LIN {X 0,Y 525.412,Z 540.645,A -85,B 0,C 180,E1 -4783.365,E2 -4783.365} C_VEL
LIN {X 0,Y 525.537,Z 527.651,A -85,B 0,C 180,E1 -4783.657,E2 -4783.657} C_VEL
LIN {X 0,Y 525.786,Z 431.838,A -85,B 0,C 180,E1 -4784.981,E2 -4784.981} C_VEL
LIN {X 0,Y 524.311,Z 422.453,A -85,B 0,C 180,E1 -4785.165,E2 -4785.165} C_VEL
LIN {X 0,Y 524.738,Z 402.773,A -85,B 0,C 180,E1 -4788.305,E2 -4788.305} C_VEL
LIN {X 0,Y 525.21,Z 383.773,A -85,B 0,C 180,E1 -4791.385,E2 -4791.385} C_VEL
LIN {X 0,Y 525.337,Z 376.275,A -85,B 0,C 180,E1 -4792.618,E2 -4792.618} C_VEL
LIN {X 0,Y 523.946,Z 368.721,A -85,B 0,C 180,E1 -4793.942,E2 -4793.942} C_VEL
LIN {X 0,Y 523.978,Z 368.713,A -85,B 0,C 180,E1 -4796.271,E2 -4796.271} C_VEL
LIN {X 0,Y 523.958,Z 368.72,A -85,B 0,C 180,E1 -4799.324,E2 -4799.324} C_VEL
LIN {X 0,Y 523.943,Z 368.716,A -85,B 0,C 180,E1 -4802.449,E2 -4802.449} C_VEL
LIN {X 0,Y 523.927,Z 368.724,A -85,B 0,C 180,E1 -4805.226,E2 -4805.226} C_VEL
LIN {X 0,Y 523.919,Z 368.718,A -85,B 0,C 180,E1 -4808.102,E2 -4808.102} C_VEL
LIN {X 0,Y 523.961,Z 368.717,A -85,B 0,C 180,E1 -4811.311,E2 -4811.311} C_VEL
LIN {X 0,Y 523.959,Z 368.719,A -85,B 0,C 180,E1 -4814.691,E2 -4814.691} C_VEL
LIN {X 0,Y 523.959,Z 368.713,A -85,B 0,C 180,E1 -4817.882,E2 -4817.882} C_VEL
LIN {X 0,Y 523.923,Z 368.725,A -85,B 0,C 180,E1 -4820.915,E2 -4820.915} C_VEL
LIN {X 0,Y 523.902,Z 368.72,A -85,B 0,C 180,E1 -4823.825,E2 -4823.825} C_VEL
LIN {X 0,Y 523.944,Z 368.723,A -85,B 0,C 180,E1 -4826.636,E2 -4826.636} C_VEL
LIN {X 0,Y 523.958,Z 368.714,A -85,B 0,C 180,E1 -4829.356,E2 -4829.356} C_VEL
LIN {X 0,Y 523.981,Z 368.714,A -85,B 0,C 180,E1 -4832.281,E2 -4832.281} C_VEL
LIN {X 0,Y 523.951,Z 368.723,A -85,B 0,C 180,E1 -4834.581,E2 -4834.581} C_VEL
LIN {X 0,Y 523.922,Z 368.718,A -85,B 0,C 180,E1 -4837.756,E2 -4837.756} C_VEL
LIN {X 0,Y 523.978,Z 368.718,A -85,B 0,C 180,E1 -4840.408,E2 -4840.408} C_VEL
LIN {X 0,Y 523.97,Z 368.716,A -85,B 0,C 180,E1 -4842.837,E2 -4842.837} C_VEL
LIN {X 0,Y 523.98,Z 368.711,A -85,B 0,C 180,E1 -4845.236,E2 -4845.236} C_VEL
LIN {X 0,Y 524.019,Z 368.715,A -85,B 0,C 180,E1 -4848.394,E2 -4848.394} C_VEL
LIN {X 0,Y 523.993,Z 368.709,A -85,B 0,C 180,E1 -4851.516,E2 -4851.516} C_VEL
LIN {X 0,Y 524.048,Z 368.705,A -85,B 0,C 180,E1 -4853.841,E2 -4853.841} C_VEL
LIN {X 0,Y 524.075,Z 368.7,A -85,B 0,C 180,E1 -4856.925,E2 -4856.925} C_VEL
LIN {X 0,Y 524.119,Z 368.699,A -85,B 0,C 180,E1 -4860,E2 -4860} C_VEL
LIN {X 0,Y 524.076,Z 368.699,A -85,B 0,C 180,E1 -4863.075,E2 -4863.075} C_VEL
LIN {X 0,Y 524.05,Z 368.711,A -85,B 0,C 180,E1 -4866.159,E2 -4866.159} C_VEL
LIN {X 0,Y 524.005,Z 368.711,A -85,B 0,C 180,E1 -4868.484,E2 -4868.484} C_VEL
LIN {X 0,Y 524.007,Z 368.712,A -85,B 0,C 180,E1 -4871.74,E2 -4871.74} C_VEL
LIN {X 0,Y 523.997,Z 368.708,A -85,B 0,C 180,E1 -4875.052,E2 -4875.052} C_VEL
LIN {X 0,Y 523.968,Z 368.721,A -85,B 0,C 180,E1 -4877.969,E2 -4877.969} C_VEL
LIN {X 0,Y 523.976,Z 368.713,A -85,B 0,C 180,E1 -4880.41,E2 -4880.41} C_VEL
LIN {X 0,Y 523.921,Z 368.718,A -85,B 0,C 180,E1 -4882.893,E2 -4882.893} C_VEL
LIN {X 0,Y 523.957,Z 368.717,A -85,B 0,C 180,E1 -4885.419,E2 -4885.419} C_VEL
LIN {X 0,Y 523.973,Z 368.717,A -85,B 0,C 180,E1 -4887.999,E2 -4887.999} C_VEL
LIN {X 0,Y 523.948,Z 368.715,A -85,B 0,C 180,E1 -4890.855,E2 -4890.855} C_VEL
LIN {X 0,Y 523.964,Z 368.721,A -85,B 0,C 180,E1 -4893.735,E2 -4893.735} C_VEL
LIN {X 0,Y 523.925,Z 368.718,A -85,B 0,C 180,E1 -4896.404,E2 -4896.404} C_VEL
LIN {X 0,Y 523.923,Z 368.72,A -85,B 0,C 180,E1 -4899.085,E2 -4899.085} C_VEL
LIN {X 0,Y 523.959,Z 368.715,A -85,B 0,C 180,E1 -4902.119,E2 -4902.119} C_VEL
LIN {X 0,Y 523.959,Z 368.719,A -85,B 0,C 180,E1 -4905.309,E2 -4905.309} C_VEL
LIN {X 0,Y 523.922,Z 368.719,A -85,B 0,C 180,E1 -4906.911,E2 -4906.911} C_VEL
LIN {X 0,Y 523.255,Z 368.809,A -85,B 0,C 180,E1 -4907.553,E2 -4907.553} C_VEL
LIN {X 0,Y 520.412,Z 369.16,A -85,B 0,C 180,E1 -4908.594,E2 -4908.594} C_VEL
LIN {X 0,Y 518.007,Z 369.464,A -85,B 0,C 180,E1 -4909.433,E2 -4909.433} C_VEL
LIN {X 0,Y 516.971,Z 369.585,A -85,B 0,C 180,E1 -4910.081,E2 -4910.081} C_VEL
LIN {X 0,Y 516.885,Z 369.595,A -85,B 0,C 180,E1 -4910.3,E2 -4910.3} C_VEL
LIN {X 0,Y 516.888,Z 369.603,A -85,B 0,C 180,E1 -4913.342,E2 -4913.342} C_VEL
LIN {X 0,Y 516.916,Z 369.591,A -85,B 0,C 180,E1 -4916.121,E2 -4916.121} C_VEL
LIN {X 0,Y 516.894,Z 369.597,A -85,B 0,C 180,E1 -4918.936,E2 -4918.936} C_VEL
LIN {X 0,Y 516.922,Z 369.594,A -85,B 0,C 180,E1 -4921.585,E2 -4921.585} C_VEL
LIN {X 0,Y 516.935,Z 369.59,A -85,B 0,C 180,E1 -4924.211,E2 -4924.211} C_VEL
LIN {X 0,Y 516.868,Z 369.603,A -85,B 0,C 180,E1 -4926.776,E2 -4926.776} C_VEL
LIN {X 0,Y 516.944,Z 369.671,A -85,B 0,C 180,E1 -4928.857,E2 -4928.857} C_VEL
LIN {X 0,Y 517.824,Z 376.138,A -85,B 0,C 180,E1 -4930.166,E2 -4930.166} C_VEL
LIN {X 0,Y 517.497,Z 389.927,A -85,B 0,C 180,E1 -4932.82,E2 -4932.82} C_VEL
LIN {X 0,Y 517.281,Z 399.757,A -85,B 0,C 180,E1 -4934.685,E2 -4934.685} C_VEL
LIN {X 0,Y 519.14,Z 410.322,A -85,B 0,C 180,E1 -4934.899,E2 -4934.899} C_VEL
LIN {X 0,Y 518.727,Z 506.835,A -85,B 0,C 180,E1 -4936.26,E2 -4936.26} C_VEL
LIN {X 0,Y 518.465,Z 520.01,A -85,B 0,C 180,E1 -4936.602,E2 -4936.602} C_VEL
LIN {X 0,Y 518.198,Z 532.106,A -85,B 0,C 180,E1 -4937.069,E2 -4937.069} C_VEL
LIN {X 0,Y 517.99,Z 543.446,A -85,B 0,C 180,E1 -4937.658,E2 -4937.658} C_VEL
LIN {X 0,Y 517.648,Z 555.196,A -85,B 0,C 180,E1 -4938.448,E2 -4938.448} C_VEL
LIN {X 0,Y 517.328,Z 565.677,A -85,B 0,C 180,E1 -4939.333,E2 -4939.333} C_VEL
LIN {X 0,Y 517.077,Z 574.24,A -85,B 0,C 180,E1 -4940.218,E2 -4940.218} C_VEL
LIN {X 0,Y 516.854,Z 582.127,A -85,B 0,C 180,E1 -4941.201,E2 -4941.201} C_VEL
LIN {X 0,Y 516.62,Z 589.84,A -85,B 0,C 180,E1 -4942.378,E2 -4942.378} C_VEL
LIN {X 0,Y 516.458,Z 596.913,A -85,B 0,C 180,E1 -4943.75,E2 -4943.75} C_VEL
LIN {X 0,Y 516.314,Z 601.629,A -85,B 0,C 180,E1 -4944.924,E2 -4944.924} C_VEL
LIN {X 0,Y 516.373,Z 605.238,A -85,B 0,C 180,E1 -4946.098,E2 -4946.098} C_VEL
LIN {X 0,Y 516.282,Z 607.106,A -85,B 0,C 180,E1 -4946.879,E2 -4946.879} C_VEL
LIN {X 0,Y 516.261,Z 608.515,A -85,B 0,C 180,E1 -4947.66,E2 -4947.66} C_VEL
LIN {X 0,Y 516.16,Z 610.136,A -85,B 0,C 180,E1 -4949.22,E2 -4949.22} C_VEL
LIN {X 0,Y 516.155,Z 610.373,A -85,B 0,C 180,E1 -4950,E2 -4950} C_VEL
LIN {X 0,Y 516.16,Z 610.19,A -85,B 0,C 180,E1 -4950.78,E2 -4950.78} C_VEL
LIN {X 0,Y 516.262,Z 608.641,A -85,B 0,C 180,E1 -4952.341,E2 -4952.341} C_VEL
LIN {X 0,Y 516.283,Z 607.286,A -85,B 0,C 180,E1 -4953.122,E2 -4953.122} C_VEL
LIN {X 0,Y 516.363,Z 604.421,A -85,B 0,C 180,E1 -4954.293,E2 -4954.293} C_VEL
LIN {X 0,Y 516.404,Z 600.537,A -85,B 0,C 180,E1 -4955.467,E2 -4955.467} C_VEL
LIN {X 0,Y 516.488,Z 594.693,A -85,B 0,C 180,E1 -4956.812,E2 -4956.812} C_VEL
LIN {X 0,Y 516.669,Z 587.996,A -85,B 0,C 180,E1 -4958.015,E2 -4958.015} C_VEL
LIN {X 0,Y 516.863,Z 579.842,A -85,B 0,C 180,E1 -4959.194,E2 -4959.194} C_VEL
LIN {X 0,Y 517.107,Z 571.496,A -85,B 0,C 180,E1 -4960.177,E2 -4960.177} C_VEL
LIN {X 0,Y 517.464,Z 561.192,A -85,B 0,C 180,E1 -4961.16,E2 -4961.16} C_VEL
LIN {X 0,Y 517.783,Z 549.377,A -85,B 0,C 180,E1 -4962.059,E2 -4962.059} C_VEL
LIN {X 0,Y 518.085,Z 538.006,A -85,B 0,C 180,E1 -4962.735,E2 -4962.735} C_VEL
LIN {X 0,Y 518.364,Z 525.984,A -85,B 0,C 180,E1 -4963.276,E2 -4963.276} C_VEL
LIN {X 0,Y 518.577,Z 512.904,A -85,B 0,C 180,E1 -4963.695,E2 -4963.695} C_VEL
LIN {X 0,Y 518.752,Z 500.391,A -85,B 0,C 180,E1 -4963.94,E2 -4963.94} C_VEL
LIN {X 0,Y 519.037,Z 409.84,A -85,B 0,C 180,E1 -4965.201,E2 -4965.201} C_VEL
LIN {X 0,Y 517.246,Z 399.719,A -85,B 0,C 180,E1 -4965.413,E2 -4965.413} C_VEL
LIN {X 0,Y 517.654,Z 384.021,A -85,B 0,C 180,E1 -4968.401,E2 -4968.401} C_VEL
LIN {X 0,Y 517.769,Z 374.986,A -85,B 0,C 180,E1 -4970.152,E2 -4970.152} C_VEL
LIN {X 0,Y 516.939,Z 369.596,A -85,B 0,C 180,E1 -4971.274,E2 -4971.274} C_VEL
LIN {X 0,Y 516.901,Z 369.6,A -85,B 0,C 180,E1 -4974.361,E2 -4974.361} C_VEL
LIN {X 0,Y 516.928,Z 369.597,A -85,B 0,C 180,E1 -4976.658,E2 -4976.658} C_VEL
LIN {X 0,Y 516.915,Z 369.591,A -85,B 0,C 180,E1 -4979.524,E2 -4979.524} C_VEL
LIN {X 0,Y 516.9,Z 369.598,A -85,B 0,C 180,E1 -4982.543,E2 -4982.543} C_VEL
LIN {X 0,Y 516.873,Z 369.597,A -85,B 0,C 180,E1 -4985.33,E2 -4985.33} C_VEL
LIN {X 0,Y 516.885,Z 369.595,A -85,B 0,C 180,E1 -4987.943,E2 -4987.943} C_VEL
LIN {X 0,Y 516.887,Z 369.602,A -85,B 0,C 180,E1 -4990.742,E2 -4990.742} C_VEL
LIN {X 0,Y 516.887,Z 369.6,A -85,B 0,C 180,E1 -4992.832,E2 -4992.832} C_VEL
LIN {X 0,Y 516.928,Z 369.592,A -85,B 0,C 180,E1 -4995.01,E2 -4995.01} C_VEL
LIN {X 0,Y 516.921,Z 369.597,A -85,B 0,C 180,E1 -4998.399,E2 -4998.399} C_VEL
LIN {X 0,Y 516.885,Z 369.595,A -85,B 0,C 180,E1 -5001.284,E2 -5001.284} C_VEL
LIN {X 0,Y 516.876,Z 369.602,A -85,B 0,C 180,E1 -5004.22,E2 -5004.22} C_VEL
LIN {X 0,Y 516.9,Z 369.593,A -85,B 0,C 180,E1 -5007.053,E2 -5007.053} C_VEL
LIN {X 0,Y 516.897,Z 369.595,A -85,B 0,C 180,E1 -5009.796,E2 -5009.796} C_VEL
LIN {X 0,Y 516.934,Z 369.595,A -85,B 0,C 180,E1 -5012.468,E2 -5012.468} C_VEL
LIN {X 0,Y 516.881,Z 369.595,A -85,B 0,C 180,E1 -5015.07,E2 -5015.07} C_VEL
LIN {X 0,Y 516.874,Z 369.597,A -85,B 0,C 180,E1 -5017.622,E2 -5017.622} C_VEL
LIN {X 0,Y 516.938,Z 369.597,A -85,B 0,C 180,E1 -5020.13,E2 -5020.13} C_VEL
LIN {X 0,Y 516.935,Z 369.591,A -85,B 0,C 180,E1 -5022.596,E2 -5022.596} C_VEL
LIN {X 0,Y 516.949,Z 369.586,A -85,B 0,C 180,E1 -5025.03,E2 -5025.03} C_VEL
LIN {X 0,Y 516.972,Z 369.589,A -85,B 0,C 180,E1 -5028.234,E2 -5028.234} C_VEL
LIN {X 0,Y 516.972,Z 369.585,A -85,B 0,C 180,E1 -5031.4,E2 -5031.4} C_VEL
LIN {X 0,Y 517.017,Z 369.584,A -85,B 0,C 180,E1 -5033.757,E2 -5033.757} C_VEL
LIN {X 0,Y 517.089,Z 369.575,A -85,B 0,C 180,E1 -5037.663,E2 -5037.663} C_VEL
LIN {X 0,Y 517.099,Z 369.568,A -85,B 0,C 180,E1 -5040.779,E2 -5040.779} C_VEL
LIN {X 0,Y 517.019,Z 369.579,A -85,B 0,C 180,E1 -5043.117,E2 -5043.117} C_VEL
LIN {X 0,Y 517.016,Z 369.58,A -85,B 0,C 180,E1 -5046.243,E2 -5046.243} C_VEL
LIN {X 0,Y 516.947,Z 369.591,A -85,B 0,C 180,E1 -5049.389,E2 -5049.389} C_VEL
LIN {X 0,Y 516.99,Z 369.588,A -85,B 0,C 180,E1 -5051.824,E2 -5051.824} C_VEL
LIN {X 0,Y 516.95,Z 369.589,A -85,B 0,C 180,E1 -5055.146,E2 -5055.146} C_VEL
LIN {X 0,Y 516.93,Z 369.59,A -85,B 0,C 180,E1 -5058.222,E2 -5058.222} C_VEL
LIN {X 0,Y 516.918,Z 369.591,A -85,B 0,C 180,E1 -5060.701,E2 -5060.701} C_VEL
LIN {X 0,Y 516.896,Z 369.594,A -85,B 0,C 180,E1 -5064.073,E2 -5064.073} C_VEL
LIN {X 0,Y 516.927,Z 369.59,A -85,B 0,C 180,E1 -5066.658,E2 -5066.658} C_VEL
LIN {X 0,Y 516.916,Z 369.597,A -85,B 0,C 180,E1 -5069.524,E2 -5069.524} C_VEL
LIN {X 0,Y 516.899,Z 369.593,A -85,B 0,C 180,E1 -5072.543,E2 -5072.543} C_VEL
LIN {X 0,Y 516.87,Z 369.604,A -85,B 0,C 180,E1 -5075.329,E2 -5075.329} C_VEL
LIN {X 0,Y 516.884,Z 369.595,A -85,B 0,C 180,E1 -5077.943,E2 -5077.943} C_VEL
LIN {X 0,Y 516.887,Z 369.597,A -85,B 0,C 180,E1 -5080.741,E2 -5080.741} C_VEL
LIN {X 0,Y 516.888,Z 369.599,A -85,B 0,C 180,E1 -5082.831,E2 -5082.831} C_VEL
LIN {X 0,Y 516.927,Z 369.597,A -85,B 0,C 180,E1 -5085.01,E2 -5085.01} C_VEL
LIN {X 0,Y 516.917,Z 369.591,A -85,B 0,C 180,E1 -5088.399,E2 -5088.399} C_VEL
LIN {X 0,Y 516.887,Z 369.599,A -85,B 0,C 180,E1 -5091.284,E2 -5091.284} C_VEL
LIN {X 0,Y 516.877,Z 369.596,A -85,B 0,C 180,E1 -5094.22,E2 -5094.22} C_VEL
LIN {X 0,Y 516.899,Z 369.6,A -85,B 0,C 180,E1 -5097.053,E2 -5097.053} C_VEL
LIN {X 0,Y 516.897,Z 369.595,A -85,B 0,C 180,E1 -5099.796,E2 -5099.796} C_VEL
LIN {X 0,Y 516.93,Z 369.595,A -85,B 0,C 180,E1 -5102.467,E2 -5102.467} C_VEL
LIN {X 0,Y 516.915,Z 369.599,A -85,B 0,C 180,E1 -5105.072,E2 -5105.072} C_VEL
LIN {X 0,Y 516.937,Z 369.68,A -85,B 0,C 180,E1 -5105.903,E2 -5105.903} C_VEL
LIN {X 0,Y 518.386,Z 377.827,A -85,B 0,C 180,E1 -5107.347,E2 -5107.347} C_VEL
LIN {X 0,Y 518.003,Z 392.507,A -85,B 0,C 180,E1 -5109.779,E2 -5109.779} C_VEL
LIN {X 0,Y 517.548,Z 409.894,A -85,B 0,C 180,E1 -5112.617,E2 -5112.617} C_VEL
LIN {X 0,Y 517.281,Z 422.435,A -85,B 0,C 180,E1 -5114.637,E2 -5114.637} C_VEL
LIN {X 0,Y 519.093,Z 434.313,A -85,B 0,C 180,E1 -5114.858,E2 -5114.858} C_VEL
LIN {X 0,Y 518.625,Z 530.314,A -85,B 0,C 180,E1 -5116.207,E2 -5116.207} C_VEL
LIN {X 0,Y 518.38,Z 543.601,A -85,B 0,C 180,E1 -5116.55,E2 -5116.55} C_VEL
LIN {X 0,Y 518.099,Z 556.895,A -85,B 0,C 180,E1 -5117.066,E2 -5117.066} C_VEL
LIN {X 0,Y 517.761,Z 569.186,A -85,B 0,C 180,E1 -5117.727,E2 -5117.727} C_VEL
LIN {X 0,Y 517.518,Z 580.946,A -85,B 0,C 180,E1 -5118.544,E2 -5118.544} C_VEL
LIN {X 0,Y 517.192,Z 591.138,A -85,B 0,C 180,E1 -5119.429,E2 -5119.429} C_VEL
LIN {X 0,Y 516.929,Z 600.309,A -85,B 0,C 180,E1 -5120.413,E2 -5120.413} C_VEL
LIN {X 0,Y 516.669,Z 609.245,A -85,B 0,C 180,E1 -5121.591,E2 -5121.591} C_VEL
LIN {X 0,Y 516.51,Z 616.437,A -85,B 0,C 180,E1 -5122.769,E2 -5122.769} C_VEL
LIN {X 0,Y 516.435,Z 622.987,A -85,B 0,C 180,E1 -5124.142,E2 -5124.142} C_VEL
LIN {X 0,Y 516.271,Z 627.317,A -85,B 0,C 180,E1 -5125.315,E2 -5125.315} C_VEL
LIN {X 0,Y 516.352,Z 629.613,A -85,B 0,C 180,E1 -5126.098,E2 -5126.098} C_VEL
LIN {X 0,Y 516.282,Z 631.47,A -85,B 0,C 180,E1 -5126.878,E2 -5126.878} C_VEL
LIN {X 0,Y 516.261,Z 632.864,A -85,B 0,C 180,E1 -5127.659,E2 -5127.659} C_VEL
LIN {X 0,Y 516.16,Z 634.463,A -85,B 0,C 180,E1 -5129.22,E2 -5129.22} C_VEL
LIN {X 0,Y 516.154,Z 634.679,A -85,B 0,C 180,E1 -5130,E2 -5130} C_VEL
LIN {X 0,Y 516.192,Z 633.859,A -85,B 0,C 180,E1 -5131.56,E2 -5131.56} C_VEL
LIN {X 0,Y 516.26,Z 632.867,A -85,B 0,C 180,E1 -5132.34,E2 -5132.34} C_VEL
LIN {X 0,Y 516.282,Z 631.474,A -85,B 0,C 180,E1 -5133.121,E2 -5133.121} C_VEL
LIN {X 0,Y 516.313,Z 628.544,A -85,B 0,C 180,E1 -5134.293,E2 -5134.293} C_VEL
LIN {X 0,Y 516.402,Z 624.578,A -85,B 0,C 180,E1 -5135.467,E2 -5135.467} C_VEL
LIN {X 0,Y 516.476,Z 618.708,A -85,B 0,C 180,E1 -5136.793,E2 -5136.793} C_VEL
LIN {X 0,Y 516.631,Z 611.806,A -85,B 0,C 180,E1 -5138.015,E2 -5138.015} C_VEL
LIN {X 0,Y 516.827,Z 603.53,A -85,B 0,C 180,E1 -5139.194,E2 -5139.194} C_VEL
LIN {X 0,Y 517.071,Z 595.048,A -85,B 0,C 180,E1 -5140.177,E2 -5140.177} C_VEL
LIN {X 0,Y 517.381,Z 584.566,A -85,B 0,C 180,E1 -5141.161,E2 -5141.161} C_VEL
LIN {X 0,Y 517.684,Z 573.343,A -85,B 0,C 180,E1 -5142.008,E2 -5142.008} C_VEL
LIN {X 0,Y 518.001,Z 562.828,A -85,B 0,C 180,E1 -5142.637,E2 -5142.637} C_VEL
LIN {X 0,Y 518.253,Z 551.168,A -85,B 0,C 180,E1 -5143.179,E2 -5143.179} C_VEL
LIN {X 0,Y 518.509,Z 538.647,A -85,B 0,C 180,E1 -5143.596,E2 -5143.596} C_VEL
LIN {X 0,Y 518.679,Z 525.979,A -85,B 0,C 180,E1 -5143.867,E2 -5143.867} C_VEL
LIN {X 0,Y 518.98,Z 432.986,A -85,B 0,C 180,E1 -5145.164,E2 -5145.164} C_VEL
LIN {X 0,Y 517.307,Z 422.331,A -85,B 0,C 180,E1 -5145.367,E2 -5145.367} C_VEL
LIN {X 0,Y 517.752,Z 402.38,A -85,B 0,C 180,E1 -5148.602,E2 -5148.602} C_VEL
LIN {X 0,Y 518.268,Z 384.883,A -85,B 0,C 180,E1 -5151.477,E2 -5151.477} C_VEL
LIN {X 0,Y 518.347,Z 377.066,A -85,B 0,C 180,E1 -5152.783,E2 -5152.783} C_VEL
LIN {X 0,Y 516.923,Z 369.596,A -85,B 0,C 180,E1 -5154.124,E2 -5154.124} C_VEL
LIN {X 0,Y 516.929,Z 369.593,A -85,B 0,C 180,E1 -5156.658,E2 -5156.658} C_VEL
LIN {X 0,Y 516.914,Z 369.594,A -85,B 0,C 180,E1 -5159.524,E2 -5159.524} C_VEL
LIN {X 0,Y 516.903,Z 369.594,A -85,B 0,C 180,E1 -5162.544,E2 -5162.544} C_VEL
LIN {X 0,Y 516.873,Z 369.601,A -85,B 0,C 180,E1 -5165.33,E2 -5165.33} C_VEL
LIN {X 0,Y 516.884,Z 369.595,A -85,B 0,C 180,E1 -5167.943,E2 -5167.943} C_VEL
LIN {X 0,Y 516.887,Z 369.6,A -85,B 0,C 180,E1 -5170.741,E2 -5170.741} C_VEL
LIN {X 0,Y 516.886,Z 369.602,A -85,B 0,C 180,E1 -5172.831,E2 -5172.831} C_VEL
LIN {X 0,Y 516.925,Z 369.597,A -85,B 0,C 180,E1 -5175.01,E2 -5175.01} C_VEL
LIN {X 0,Y 516.919,Z 369.593,A -85,B 0,C 180,E1 -5178.398,E2 -5178.398} C_VEL
LIN {X 0,Y 516.883,Z 369.597,A -85,B 0,C 180,E1 -5181.284,E2 -5181.284} C_VEL
LIN {X 0,Y 516.873,Z 369.598,A -85,B 0,C 180,E1 -5184.22,E2 -5184.22} C_VEL
LIN {X 0,Y 516.897,Z 369.597,A -85,B 0,C 180,E1 -5187.053,E2 -5187.053} C_VEL
LIN {X 0,Y 516.895,Z 369.593,A -85,B 0,C 180,E1 -5189.796,E2 -5189.796} C_VEL
LIN {X 0,Y 516.931,Z 369.595,A -85,B 0,C 180,E1 -5192.467,E2 -5192.467} C_VEL
LIN {X 0,Y 516.879,Z 369.598,A -85,B 0,C 180,E1 -5195.07,E2 -5195.07} C_VEL
LIN {X 0,Y 516.871,Z 369.596,A -85,B 0,C 180,E1 -5197.622,E2 -5197.622} C_VEL
LIN {X 0,Y 516.935,Z 369.592,A -85,B 0,C 180,E1 -5200.13,E2 -5200.13} C_VEL
LIN {X 0,Y 516.924,Z 369.597,A -85,B 0,C 180,E1 -5202.596,E2 -5202.596} C_VEL
LIN {X 0,Y 516.946,Z 369.588,A -85,B 0,C 180,E1 -5205.03,E2 -5205.03} C_VEL
LIN {X 0,Y 517.008,Z 369.586,A -85,B 0,C 180,E1 -5208.235,E2 -5208.235} C_VEL
LIN {X 0,Y 516.961,Z 369.585,A -85,B 0,C 180,E1 -5211.4,E2 -5211.4} C_VEL
LIN {X 0,Y 517.013,Z 369.58,A -85,B 0,C 180,E1 -5213.757,E2 -5213.757} C_VEL
LIN {X 0,Y 517.086,Z 369.571,A -85,B 0,C 180,E1 -5217.663,E2 -5217.663} C_VEL
LIN {X 0,Y 517.097,Z 369.57,A -85,B 0,C 180,E1 -5220.779,E2 -5220.779} C_VEL
LIN {X 0,Y 517.017,Z 369.578,A -85,B 0,C 180,E1 -5223.117,E2 -5223.117} C_VEL
LIN {X 0,Y 517.014,Z 369.586,A -85,B 0,C 180,E1 -5226.243,E2 -5226.243} C_VEL
LIN {X 0,Y 516.949,Z 369.587,A -85,B 0,C 180,E1 -5229.389,E2 -5229.389} C_VEL
LIN {X 0,Y 516.956,Z 369.591,A -85,B 0,C 180,E1 -5231.807,E2 -5231.807} C_VEL
LIN {X 0,Y 516.948,Z 369.587,A -85,B 0,C 180,E1 -5235.147,E2 -5235.147} C_VEL
LIN {X 0,Y 516.93,Z 369.594,A -85,B 0,C 180,E1 -5238.222,E2 -5238.222} C_VEL
LIN {X 0,Y 516.916,Z 369.591,A -85,B 0,C 180,E1 -5240.701,E2 -5240.701} C_VEL
LIN {X 0,Y 516.915,Z 369.596,A -85,B 0,C 180,E1 -5244.072,E2 -5244.072} C_VEL
LIN {X 0,Y 516.93,Z 369.589,A -85,B 0,C 180,E1 -5246.658,E2 -5246.658} C_VEL
LIN {X 0,Y 516.914,Z 369.596,A -85,B 0,C 180,E1 -5249.524,E2 -5249.524} C_VEL
LIN {X 0,Y 516.901,Z 369.593,A -85,B 0,C 180,E1 -5252.544,E2 -5252.544} C_VEL
LIN {X 0,Y 516.884,Z 369.599,A -85,B 0,C 180,E1 -5255.332,E2 -5255.332} C_VEL
LIN {X 0,Y 516.884,Z 369.599,A -85,B 0,C 180,E1 -5257.943,E2 -5257.943} C_VEL
LIN {X 0,Y 516.887,Z 369.594,A -85,B 0,C 180,E1 -5260.742,E2 -5260.742} C_VEL
LIN {X 0,Y 516.908,Z 369.592,A -85,B 0,C 180,E1 -5262.829,E2 -5262.829} C_VEL
LIN {X 0,Y 516.926,Z 369.592,A -85,B 0,C 180,E1 -5265.01,E2 -5265.01} C_VEL
LIN {X 0,Y 516.918,Z 369.59,A -85,B 0,C 180,E1 -5268.399,E2 -5268.399} C_VEL
LIN {X 0,Y 516.885,Z 369.595,A -85,B 0,C 180,E1 -5270.3,E2 -5270.3} C_VEL
LIN {X 0,Y 516.215,Z 369.682,A -85,B 0,C 180,E1 -5270.95,E2 -5270.95} C_VEL
LIN {X 0,Y 513.37,Z 370.039,A -85,B 0,C 180,E1 -5272.006,E2 -5272.006} C_VEL
LIN {X 0,Y 510.963,Z 370.341,A -85,B 0,C 180,E1 -5272.856,E2 -5272.856} C_VEL
LIN {X 0,Y 509.923,Z 370.469,A -85,B 0,C 180,E1 -5273.513,E2 -5273.513} C_VEL
LIN {X 0,Y 509.835,Z 370.476,A -85,B 0,C 180,E1 -5273.735,E2 -5273.735} C_VEL
LIN {X 0,Y 509.865,Z 370.469,A -85,B 0,C 180,E1 -5276.539,E2 -5276.539} C_VEL
LIN {X 0,Y 509.848,Z 370.479,A -85,B 0,C 180,E1 -5279.334,E2 -5279.334} C_VEL
LIN {X 0,Y 509.895,Z 370.465,A -85,B 0,C 180,E1 -5282.055,E2 -5282.055} C_VEL
LIN {X 0,Y 509.879,Z 370.472,A -85,B 0,C 180,E1 -5284.704,E2 -5284.704} C_VEL
LIN {X 0,Y 509.83,Z 370.482,A -85,B 0,C 180,E1 -5287.458,E2 -5287.458} C_VEL
LIN {X 0,Y 509.918,Z 370.601,A -85,B 0,C 180,E1 -5288.71,E2 -5288.71} C_VEL
LIN {X 0,Y 510.86,Z 377.333,A -85,B 0,C 180,E1 -5290.093,E2 -5290.093} C_VEL
LIN {X 0,Y 510.517,Z 391.131,A -85,B 0,C 180,E1 -5292.784,E2 -5292.784} C_VEL
LIN {X 0,Y 510.264,Z 399.943,A -85,B 0,C 180,E1 -5294.471,E2 -5294.471} C_VEL
LIN {X 0,Y 512.268,Z 410.948,A -85,B 0,C 180,E1 -5294.698,E2 -5294.698} C_VEL
LIN {X 0,Y 511.857,Z 507.03,A -85,B 0,C 180,E1 -5296.072,E2 -5296.072} C_VEL
LIN {X 0,Y 511.588,Z 520.195,A -85,B 0,C 180,E1 -5296.419,E2 -5296.419} C_VEL
LIN {X 0,Y 511.278,Z 532.288,A -85,B 0,C 180,E1 -5296.891,E2 -5296.891} C_VEL
LIN {X 0,Y 511.049,Z 544.291,A -85,B 0,C 180,E1 -5297.529,E2 -5297.529} C_VEL
LIN {X 0,Y 510.687,Z 555.371,A -85,B 0,C 180,E1 -5298.288,E2 -5298.288} C_VEL
LIN {X 0,Y 510.354,Z 565.851,A -85,B 0,C 180,E1 -5299.186,E2 -5299.186} C_VEL
LIN {X 0,Y 510.093,Z 574.412,A -85,B 0,C 180,E1 -5300.083,E2 -5300.083} C_VEL
LIN {X 0,Y 509.836,Z 582.298,A -85,B 0,C 180,E1 -5301.079,E2 -5301.079} C_VEL
LIN {X 0,Y 509.576,Z 590.011,A -85,B 0,C 180,E1 -5302.272,E2 -5302.272} C_VEL
LIN {X 0,Y 509.395,Z 597.083,A -85,B 0,C 180,E1 -5303.663,E2 -5303.663} C_VEL
LIN {X 0,Y 509.248,Z 601.799,A -85,B 0,C 180,E1 -5304.853,E2 -5304.853} C_VEL
LIN {X 0,Y 509.304,Z 605.406,A -85,B 0,C 180,E1 -5306.044,E2 -5306.044} C_VEL
LIN {X 0,Y 509.201,Z 607.275,A -85,B 0,C 180,E1 -5306.835,E2 -5306.835} C_VEL
LIN {X 0,Y 509.19,Z 608.683,A -85,B 0,C 180,E1 -5307.627,E2 -5307.627} C_VEL
LIN {X 0,Y 509.074,Z 610.303,A -85,B 0,C 180,E1 -5309.209,E2 -5309.209} C_VEL
LIN {X 0,Y 509.066,Z 610.54,A -85,B 0,C 180,E1 -5310,E2 -5310} C_VEL
LIN {X 0,Y 509.074,Z 610.357,A -85,B 0,C 180,E1 -5310.791,E2 -5310.791} C_VEL
LIN {X 0,Y 509.19,Z 608.806,A -85,B 0,C 180,E1 -5312.373,E2 -5312.373} C_VEL
LIN {X 0,Y 509.202,Z 607.452,A -85,B 0,C 180,E1 -5313.165,E2 -5313.165} C_VEL
LIN {X 0,Y 509.284,Z 604.586,A -85,B 0,C 180,E1 -5314.353,E2 -5314.353} C_VEL
LIN {X 0,Y 509.346,Z 600.702,A -85,B 0,C 180,E1 -5315.543,E2 -5315.543} C_VEL
LIN {X 0,Y 509.413,Z 595.692,A -85,B 0,C 180,E1 -5316.734,E2 -5316.734} C_VEL
LIN {X 0,Y 509.61,Z 589.382,A -85,B 0,C 180,E1 -5317.927,E2 -5317.927} C_VEL
LIN {X 0,Y 509.802,Z 581.485,A -85,B 0,C 180,E1 -5319.122,E2 -5319.122} C_VEL
LIN {X 0,Y 510.089,Z 573.432,A -85,B 0,C 180,E1 -5320.118,E2 -5320.118} C_VEL
LIN {X 0,Y 510.411,Z 563.606,A -85,B 0,C 180,E1 -5321.115,E2 -5321.115} C_VEL
LIN {X 0,Y 510.723,Z 553.942,A -85,B 0,C 180,E1 -5321.912,E2 -5321.912} C_VEL
LIN {X 0,Y 511.042,Z 543.025,A -85,B 0,C 180,E1 -5322.638,E2 -5322.638} C_VEL
LIN {X 0,Y 511.327,Z 530.914,A -85,B 0,C 180,E1 -5323.26,E2 -5323.26} C_VEL
LIN {X 0,Y 511.612,Z 518.336,A -85,B 0,C 180,E1 -5323.733,E2 -5323.733} C_VEL
LIN {X 0,Y 511.857,Z 505.087,A -85,B 0,C 180,E1 -5324.055,E2 -5324.055} C_VEL
LIN {X 0,Y 512.165,Z 410.484,A -85,B 0,C 180,E1 -5325.402,E2 -5325.402} C_VEL
LIN {X 0,Y 510.261,Z 399.864,A -85,B 0,C 180,E1 -5325.631,E2 -5325.631} C_VEL
LIN {X 0,Y 510.723,Z 384.154,A -85,B 0,C 180,E1 -5328.66,E2 -5328.66} C_VEL
LIN {X 0,Y 510.759,Z 375.521,A -85,B 0,C 180,E1 -5330.361,E2 -5330.361} C_VEL
LIN {X 0,Y 509.887,Z 370.475,A -85,B 0,C 180,E1 -5331.424,E2 -5331.424} C_VEL
LIN {X 0,Y 509.859,Z 370.479,A -85,B 0,C 180,E1 -5334.528,E2 -5334.528} C_VEL
LIN {X 0,Y 509.887,Z 370.474,A -85,B 0,C 180,E1 -5337.056,E2 -5337.056} C_VEL
LIN {X 0,Y 509.862,Z 370.469,A -85,B 0,C 180,E1 -5339.751,E2 -5339.751} C_VEL
LIN {X 0,Y 509.877,Z 370.476,A -85,B 0,C 180,E1 -5342.774,E2 -5342.774} C_VEL
LIN {X 0,Y 509.832,Z 370.473,A -85,B 0,C 180,E1 -5345.579,E2 -5345.579} C_VEL
LIN {X 0,Y 509.854,Z 370.474,A -85,B 0,C 180,E1 -5348.338,E2 -5348.338} C_VEL
LIN {X 0,Y 509.859,Z 370.47,A -85,B 0,C 180,E1 -5351.426,E2 -5351.426} C_VEL
LIN {X 0,Y 509.861,Z 370.477,A -85,B 0,C 180,E1 -5354.668,E2 -5354.668} C_VEL
LIN {X 0,Y 509.865,Z 370.472,A -85,B 0,C 180,E1 -5358.103,E2 -5358.103} C_VEL
LIN {X 0,Y 509.85,Z 370.477,A -85,B 0,C 180,E1 -5360.648,E2 -5360.648} C_VEL
LIN {X 0,Y 509.829,Z 370.474,A -85,B 0,C 180,E1 -5363.647,E2 -5363.647} C_VEL
LIN {X 0,Y 509.864,Z 370.475,A -85,B 0,C 180,E1 -5366.539,E2 -5366.539} C_VEL
LIN {X 0,Y 509.851,Z 370.471,A -85,B 0,C 180,E1 -5369.334,E2 -5369.334} C_VEL
LIN {X 0,Y 509.899,Z 370.47,A -85,B 0,C 180,E1 -5372.055,E2 -5372.055} C_VEL
LIN {X 0,Y 509.846,Z 370.474,A -85,B 0,C 180,E1 -5374.702,E2 -5374.702} C_VEL
LIN {X 0,Y 509.832,Z 370.474,A -85,B 0,C 180,E1 -5377.458,E2 -5377.458} C_VEL
LIN {X 0,Y 509.923,Z 370.466,A -85,B 0,C 180,E1 -5379.845,E2 -5379.845} C_VEL
LIN {X 0,Y 509.89,Z 370.466,A -85,B 0,C 180,E1 -5383.175,E2 -5383.175} C_VEL
LIN {X 0,Y 509.87,Z 370.471,A -85,B 0,C 180,E1 -5385.634,E2 -5385.634} C_VEL
LIN {X 0,Y 509.919,Z 370.462,A -85,B 0,C 180,E1 -5388.875,E2 -5388.875} C_VEL
LIN {X 0,Y 509.957,Z 370.465,A -85,B 0,C 180,E1 -5392.078,E2 -5392.078} C_VEL
LIN {X 0,Y 509.987,Z 370.456,A -85,B 0,C 180,E1 -5394.464,E2 -5394.464} C_VEL
LIN {X 0,Y 510.06,Z 370.45,A -85,B 0,C 180,E1 -5397.631,E2 -5397.631} C_VEL
LIN {X 0,Y 510.069,Z 370.443,A -85,B 0,C 180,E1 -5400.789,E2 -5400.789} C_VEL
LIN {X 0,Y 509.961,Z 370.458,A -85,B 0,C 180,E1 -5403.16,E2 -5403.16} C_VEL
LIN {X 0,Y 509.985,Z 370.455,A -85,B 0,C 180,E1 -5406.33,E2 -5406.33} C_VEL
LIN {X 0,Y 509.888,Z 370.473,A -85,B 0,C 180,E1 -5409.521,E2 -5409.521} C_VEL
LIN {X 0,Y 509.957,Z 370.462,A -85,B 0,C 180,E1 -5411.93,E2 -5411.93} C_VEL
LIN {X 0,Y 509.9,Z 370.469,A -85,B 0,C 180,E1 -5415.242,E2 -5415.242} C_VEL
LIN {X 0,Y 509.887,Z 370.469,A -85,B 0,C 180,E1 -5417.998,E2 -5417.998} C_VEL
LIN {X 0,Y 509.856,Z 370.472,A -85,B 0,C 180,E1 -5421.001,E2 -5421.001} C_VEL
LIN {X 0,Y 509.828,Z 370.481,A -85,B 0,C 180,E1 -5423.564,E2 -5423.564} C_VEL
LIN {X 0,Y 509.915,Z 370.463,A -85,B 0,C 180,E1 -5426.378,E2 -5426.378} C_VEL
LIN {X 0,Y 509.881,Z 370.469,A -85,B 0,C 180,E1 -5428.844,E2 -5428.844} C_VEL
LIN {X 0,Y 509.825,Z 370.479,A -85,B 0,C 180,E1 -5431.59,E2 -5431.59} C_VEL
LIN {X 0,Y 509.842,Z 370.472,A -85,B 0,C 180,E1 -5434.414,E2 -5434.414} C_VEL
LIN {X 0,Y 509.82,Z 370.482,A -85,B 0,C 180,E1 -5437.341,E2 -5437.341} C_VEL
LIN {X 0,Y 509.842,Z 370.472,A -85,B 0,C 180,E1 -5440.382,E2 -5440.382} C_VEL
LIN {X 0,Y 509.829,Z 370.481,A -85,B 0,C 180,E1 -5443.062,E2 -5443.062} C_VEL
LIN {X 0,Y 509.834,Z 370.474,A -85,B 0,C 180,E1 -5445.792,E2 -5445.792} C_VEL
LIN {X 0,Y 509.859,Z 370.472,A -85,B 0,C 180,E1 -5448.574,E2 -5448.574} C_VEL
LIN {X 0,Y 509.856,Z 370.47,A -85,B 0,C 180,E1 -5451.786,E2 -5451.786} C_VEL
LIN {X 0,Y 509.837,Z 370.477,A -85,B 0,C 180,E1 -5454.622,E2 -5454.622} C_VEL
LIN {X 0,Y 509.865,Z 370.47,A -85,B 0,C 180,E1 -5457.481,E2 -5457.481} C_VEL
LIN {X 0,Y 509.862,Z 370.473,A -85,B 0,C 180,E1 -5460.273,E2 -5460.273} C_VEL
LIN {X 0,Y 509.888,Z 370.473,A -85,B 0,C 180,E1 -5462.944,E2 -5462.944} C_VEL
LIN {X 0,Y 509.925,Z 370.633,A -85,B 0,C 180,E1 -5465.739,E2 -5465.739} C_VEL
LIN {X 0,Y 511.482,Z 379.734,A -85,B 0,C 180,E1 -5467.373,E2 -5467.373} C_VEL
LIN {X 0,Y 510.992,Z 394.739,A -85,B 0,C 180,E1 -5469.889,E2 -5469.889} C_VEL
LIN {X 0,Y 510.517,Z 412.238,A -85,B 0,C 180,E1 -5472.784,E2 -5472.784} C_VEL
LIN {X 0,Y 510.255,Z 422.187,A -85,B 0,C 180,E1 -5474.418,E2 -5474.418} C_VEL
LIN {X 0,Y 512.249,Z 434.973,A -85,B 0,C 180,E1 -5474.663,E2 -5474.663} C_VEL
LIN {X 0,Y 511.745,Z 530.147,A -85,B 0,C 180,E1 -5476.017,E2 -5476.017} C_VEL
LIN {X 0,Y 511.481,Z 543.434,A -85,B 0,C 180,E1 -5476.365,E2 -5476.365} C_VEL
LIN {X 0,Y 511.158,Z 556.727,A -85,B 0,C 180,E1 -5476.887,E2 -5476.887} C_VEL
LIN {X 0,Y 510.859,Z 568.314,A -85,B 0,C 180,E1 -5477.513,E2 -5477.513} C_VEL
LIN {X 0,Y 510.581,Z 579.483,A -85,B 0,C 180,E1 -5478.286,E2 -5478.286} C_VEL
LIN {X 0,Y 510.247,Z 589.926,A -85,B 0,C 180,E1 -5479.183,E2 -5479.183} C_VEL
LIN {X 0,Y 509.959,Z 598.463,A -85,B 0,C 180,E1 -5480.08,E2 -5480.08} C_VEL
LIN {X 0,Y 509.698,Z 606.339,A -85,B 0,C 180,E1 -5481.076,E2 -5481.076} C_VEL
LIN {X 0,Y 509.508,Z 614.032,A -85,B 0,C 180,E1 -5482.271,E2 -5482.271} C_VEL
LIN {X 0,Y 509.316,Z 621.123,A -85,B 0,C 180,E1 -5483.662,E2 -5483.662} C_VEL
LIN {X 0,Y 509.248,Z 625.84,A -85,B 0,C 180,E1 -5484.853,E2 -5484.853} C_VEL
LIN {X 0,Y 509.245,Z 629.445,A -85,B 0,C 180,E1 -5486.043,E2 -5486.043} C_VEL
LIN {X 0,Y 509.2,Z 631.303,A -85,B 0,C 180,E1 -5486.835,E2 -5486.835} C_VEL
LIN {X 0,Y 509.189,Z 632.697,A -85,B 0,C 180,E1 -5487.627,E2 -5487.627} C_VEL
LIN {X 0,Y 509.073,Z 634.296,A -85,B 0,C 180,E1 -5489.209,E2 -5489.209} C_VEL
LIN {X 0,Y 509.065,Z 634.512,A -85,B 0,C 180,E1 -5490,E2 -5490} C_VEL
LIN {X 0,Y 509.112,Z 633.692,A -85,B 0,C 180,E1 -5491.582,E2 -5491.582} C_VEL
LIN {X 0,Y 509.189,Z 632.7,A -85,B 0,C 180,E1 -5492.373,E2 -5492.373} C_VEL
LIN {X 0,Y 509.2,Z 631.307,A -85,B 0,C 180,E1 -5493.165,E2 -5493.165} C_VEL
LIN {X 0,Y 509.205,Z 628.376,A -85,B 0,C 180,E1 -5494.353,E2 -5494.353} C_VEL
LIN {X 0,Y 509.317,Z 624.41,A -85,B 0,C 180,E1 -5495.543,E2 -5495.543} C_VEL
LIN {X 0,Y 509.401,Z 618.761,A -85,B 0,C 180,E1 -5496.844,E2 -5496.844} C_VEL
LIN {X 0,Y 509.561,Z 611.638,A -85,B 0,C 180,E1 -5498.127,E2 -5498.127} C_VEL
LIN {X 0,Y 509.776,Z 603.362,A -85,B 0,C 180,E1 -5499.322,E2 -5499.322} C_VEL
LIN {X 0,Y 510.048,Z 594.88,A -85,B 0,C 180,E1 -5500.319,E2 -5500.319} C_VEL
LIN {X 0,Y 510.392,Z 584.398,A -85,B 0,C 180,E1 -5501.316,E2 -5501.316} C_VEL
LIN {X 0,Y 510.698,Z 573.888,A -85,B 0,C 180,E1 -5502.124,E2 -5502.124} C_VEL
LIN {X 0,Y 511.052,Z 562.66,A -85,B 0,C 180,E1 -5502.812,E2 -5502.812} C_VEL
LIN {X 0,Y 511.325,Z 551,A -85,B 0,C 180,E1 -5503.361,E2 -5503.361} C_VEL
LIN {X 0,Y 511.622,Z 537.565,A -85,B 0,C 180,E1 -5503.808,E2 -5503.808} C_VEL
LIN {X 0,Y 511.816,Z 524.297,A -85,B 0,C 180,E1 -5504.082,E2 -5504.082} C_VEL
LIN {X 0,Y 512.177,Z 434.034,A -85,B 0,C 180,E1 -5505.353,E2 -5505.353} C_VEL
LIN {X 0,Y 510.298,Z 422.066,A -85,B 0,C 180,E1 -5505.599,E2 -5505.599} C_VEL
LIN {X 0,Y 510.755,Z 403.486,A -85,B 0,C 180,E1 -5508.658,E2 -5508.658} C_VEL
LIN {X 0,Y 511.331,Z 385.992,A -85,B 0,C 180,E1 -5511.572,E2 -5511.572} C_VEL
LIN {X 0,Y 511.332,Z 377.912,A -85,B 0,C 180,E1 -5512.944,E2 -5512.944} C_VEL
LIN {X 0,Y 509.875,Z 370.474,A -85,B 0,C 180,E1 -5514.317,E2 -5514.317} C_VEL
LIN {X 0,Y 509.888,Z 370.474,A -85,B 0,C 180,E1 -5517.055,E2 -5517.055} C_VEL
LIN {X 0,Y 509.86,Z 370.471,A -85,B 0,C 180,E1 -5519.751,E2 -5519.751} C_VEL
LIN {X 0,Y 509.88,Z 370.471,A -85,B 0,C 180,E1 -5522.775,E2 -5522.775} C_VEL
LIN {X 0,Y 509.831,Z 370.475,A -85,B 0,C 180,E1 -5525.579,E2 -5525.579} C_VEL
LIN {X 0,Y 509.853,Z 370.471,A -85,B 0,C 180,E1 -5528.338,E2 -5528.338} C_VEL
LIN {X 0,Y 509.859,Z 370.472,A -85,B 0,C 180,E1 -5531.425,E2 -5531.425} C_VEL
LIN {X 0,Y 509.859,Z 370.475,A -85,B 0,C 180,E1 -5534.668,E2 -5534.668} C_VEL
LIN {X 0,Y 509.863,Z 370.47,A -85,B 0,C 180,E1 -5538.103,E2 -5538.103} C_VEL
LIN {X 0,Y 509.848,Z 370.477,A -85,B 0,C 180,E1 -5540.648,E2 -5540.648} C_VEL
LIN {X 0,Y 509.827,Z 370.474,A -85,B 0,C 180,E1 -5543.647,E2 -5543.647} C_VEL
LIN {X 0,Y 509.861,Z 370.475,A -85,B 0,C 180,E1 -5546.539,E2 -5546.539} C_VEL
LIN {X 0,Y 509.848,Z 370.472,A -85,B 0,C 180,E1 -5549.334,E2 -5549.334} C_VEL
LIN {X 0,Y 509.897,Z 370.466,A -85,B 0,C 180,E1 -5552.055,E2 -5552.055} C_VEL
LIN {X 0,Y 509.844,Z 370.479,A -85,B 0,C 180,E1 -5554.702,E2 -5554.702} C_VEL
LIN {X 0,Y 509.829,Z 370.473,A -85,B 0,C 180,E1 -5557.458,E2 -5557.458} C_VEL
LIN {X 0,Y 509.92,Z 370.463,A -85,B 0,C 180,E1 -5559.845,E2 -5559.845} C_VEL
LIN {X 0,Y 509.885,Z 370.467,A -85,B 0,C 180,E1 -5563.175,E2 -5563.175} C_VEL
LIN {X 0,Y 509.867,Z 370.469,A -85,B 0,C 180,E1 -5565.634,E2 -5565.634} C_VEL
LIN {X 0,Y 509.925,Z 370.464,A -85,B 0,C 180,E1 -5568.875,E2 -5568.875} C_VEL
LIN {X 0,Y 509.925,Z 370.467,A -85,B 0,C 180,E1 -5572.078,E2 -5572.078} C_VEL
LIN {X 0,Y 509.984,Z 370.461,A -85,B 0,C 180,E1 -5574.464,E2 -5574.464} C_VEL
LIN {X 0,Y 510.057,Z 370.446,A -85,B 0,C 180,E1 -5577.631,E2 -5577.631} C_VEL
LIN {X 0,Y 510.067,Z 370.445,A -85,B 0,C 180,E1 -5580.79,E2 -5580.79} C_VEL
LIN {X 0,Y 509.959,Z 370.457,A -85,B 0,C 180,E1 -5583.16,E2 -5583.16} C_VEL
LIN {X 0,Y 509.982,Z 370.46,A -85,B 0,C 180,E1 -5586.33,E2 -5586.33} C_VEL
LIN {X 0,Y 509.915,Z 370.464,A -85,B 0,C 180,E1 -5588.72,E2 -5588.72} C_VEL
LIN {X 0,Y 509.908,Z 370.471,A -85,B 0,C 180,E1 -5591.932,E2 -5591.932} C_VEL
LIN {X 0,Y 509.897,Z 370.465,A -85,B 0,C 180,E1 -5595.242,E2 -5595.242} C_VEL
LIN {X 0,Y 509.892,Z 370.474,A -85,B 0,C 180,E1 -5598.001,E2 -5598.001} C_VEL
LIN {X 0,Y 509.854,Z 370.47,A -85,B 0,C 180,E1 -5601.002,E2 -5601.002} C_VEL
LIN {X 0,Y 509.841,Z 370.477,A -85,B 0,C 180,E1 -5603.563,E2 -5603.563} C_VEL
LIN {X 0,Y 509.915,Z 370.464,A -85,B 0,C 180,E1 -5606.379,E2 -5606.379} C_VEL
LIN {X 0,Y 509.88,Z 370.467,A -85,B 0,C 180,E1 -5608.844,E2 -5608.844} C_VEL
LIN {X 0,Y 509.826,Z 370.481,A -85,B 0,C 180,E1 -5611.59,E2 -5611.59} C_VEL
LIN {X 0,Y 509.856,Z 370.471,A -85,B 0,C 180,E1 -5614.413,E2 -5614.413} C_VEL
LIN {X 0,Y 509.822,Z 370.479,A -85,B 0,C 180,E1 -5617.341,E2 -5617.341} C_VEL
LIN {X 0,Y 509.841,Z 370.472,A -85,B 0,C 180,E1 -5620.382,E2 -5620.382} C_VEL
LIN {X 0,Y 509.843,Z 370.474,A -85,B 0,C 180,E1 -5623.064,E2 -5623.064} C_VEL
LIN {X 0,Y 509.834,Z 370.477,A -85,B 0,C 180,E1 -5625.792,E2 -5625.792} C_VEL
LIN {X 0,Y 509.859,Z 370.47,A -85,B 0,C 180,E1 -5628.575,E2 -5628.575} C_VEL
LIN {X 0,Y 509.855,Z 370.474,A -85,B 0,C 180,E1 -5631.786,E2 -5631.786} C_VEL
LIN {X 0,Y 509.835,Z 370.476,A -85,B 0,C 180,E1 -5633.735,E2 -5633.735} C_VEL
LIN {X 0,Y 509.17,Z 370.557,A -85,B 0,C 180,E1 -5634.395,E2 -5634.395} C_VEL
LIN {X 0,Y 506.353,Z 370.914,A -85,B 0,C 180,E1 -5635.467,E2 -5635.467} C_VEL
LIN {X 0,Y 503.96,Z 371.212,A -85,B 0,C 180,E1 -5636.33,E2 -5636.33} C_VEL
LIN {X 0,Y 502.909,Z 371.339,A -85,B 0,C 180,E1 -5636.996,E2 -5636.996} C_VEL
LIN {X 0,Y 502.811,Z 371.35,A -85,B 0,C 180,E1 -5637.222,E2 -5637.222} C_VEL
LIN {X 0,Y 502.818,Z 371.347,A -85,B 0,C 180,E1 -5640.065,E2 -5640.065} C_VEL
LIN {X 0,Y 502.835,Z 371.345,A -85,B 0,C 180,E1 -5642.533,E2 -5642.533} C_VEL
LIN {X 0,Y 502.83,Z 371.353,A -85,B 0,C 180,E1 -5645.299,E2 -5645.299} C_VEL
LIN {X 0,Y 502.837,Z 371.397,A -85,B 0,C 180,E1 -5648.53,E2 -5648.53} C_VEL
LIN {X 0,Y 503.912,Z 378.529,A -85,B 0,C 180,E1 -5650.02,E2 -5650.02} C_VEL
LIN {X 0,Y 503.518,Z 392.333,A -85,B 0,C 180,E1 -5652.746,E2 -5652.746} C_VEL
LIN {X 0,Y 503.277,Z 400.118,A -85,B 0,C 180,E1 -5654.255,E2 -5654.255} C_VEL
LIN {X 0,Y 505.444,Z 411.906,A -85,B 0,C 180,E1 -5654.497,E2 -5654.497} C_VEL
LIN {X 0,Y 504.984,Z 507.226,A -85,B 0,C 180,E1 -5655.878,E2 -5655.878} C_VEL
LIN {X 0,Y 504.696,Z 520.382,A -85,B 0,C 180,E1 -5656.23,E2 -5656.23} C_VEL
LIN {X 0,Y 504.378,Z 532.469,A -85,B 0,C 180,E1 -5656.708,E2 -5656.708} C_VEL
LIN {X 0,Y 504.142,Z 544.194,A -85,B 0,C 180,E1 -5657.337,E2 -5657.337} C_VEL
LIN {X 0,Y 503.733,Z 555.547,A -85,B 0,C 180,E1 -5658.124,E2 -5658.124} C_VEL
LIN {X 0,Y 503.386,Z 566.024,A -85,B 0,C 180,E1 -5659.034,E2 -5659.034} C_VEL
LIN {X 0,Y 503.108,Z 574.585,A -85,B 0,C 180,E1 -5659.944,E2 -5659.944} C_VEL
LIN {X 0,Y 502.816,Z 582.471,A -85,B 0,C 180,E1 -5660.953,E2 -5660.953} C_VEL
LIN {X 0,Y 502.533,Z 590.182,A -85,B 0,C 180,E1 -5662.163,E2 -5662.163} C_VEL
LIN {X 0,Y 502.324,Z 597.254,A -85,B 0,C 180,E1 -5663.574,E2 -5663.574} C_VEL
LIN {X 0,Y 502.187,Z 601.968,A -85,B 0,C 180,E1 -5664.781,E2 -5664.781} C_VEL
LIN {X 0,Y 502.218,Z 605.575,A -85,B 0,C 180,E1 -5665.988,E2 -5665.988} C_VEL
LIN {X 0,Y 502.124,Z 607.443,A -85,B 0,C 180,E1 -5666.791,E2 -5666.791} C_VEL
LIN {X 0,Y 502.121,Z 608.85,A -85,B 0,C 180,E1 -5667.594,E2 -5667.594} C_VEL
LIN {X 0,Y 501.991,Z 610.47,A -85,B 0,C 180,E1 -5669.198,E2 -5669.198} C_VEL
LIN {X 0,Y 501.981,Z 610.707,A -85,B 0,C 180,E1 -5670,E2 -5670} C_VEL
LIN {X 0,Y 501.991,Z 610.523,A -85,B 0,C 180,E1 -5670.802,E2 -5670.802} C_VEL
LIN {X 0,Y 502.121,Z 608.972,A -85,B 0,C 180,E1 -5672.407,E2 -5672.407} C_VEL
LIN {X 0,Y 502.125,Z 607.617,A -85,B 0,C 180,E1 -5673.21,E2 -5673.21} C_VEL
LIN {X 0,Y 502.19,Z 604.752,A -85,B 0,C 180,E1 -5674.415,E2 -5674.415} C_VEL
LIN {X 0,Y 502.29,Z 600.866,A -85,B 0,C 180,E1 -5675.621,E2 -5675.621} C_VEL
LIN {X 0,Y 502.354,Z 595.857,A -85,B 0,C 180,E1 -5676.829,E2 -5676.829} C_VEL
LIN {X 0,Y 502.564,Z 589.546,A -85,B 0,C 180,E1 -5678.039,E2 -5678.039} C_VEL
LIN {X 0,Y 502.777,Z 581.647,A -85,B 0,C 180,E1 -5679.251,E2 -5679.251} C_VEL
LIN {X 0,Y 503.068,Z 573.595,A -85,B 0,C 180,E1 -5680.261,E2 -5680.261} C_VEL
LIN {X 0,Y 503.457,Z 563.767,A -85,B 0,C 180,E1 -5681.27,E2 -5681.27} C_VEL
LIN {X 0,Y 503.78,Z 554.101,A -85,B 0,C 180,E1 -5682.079,E2 -5682.079} C_VEL
LIN {X 0,Y 504.11,Z 543.158,A -85,B 0,C 180,E1 -5682.816,E2 -5682.816} C_VEL
LIN {X 0,Y 504.423,Z 531.067,A -85,B 0,C 180,E1 -5683.445,E2 -5683.445} C_VEL
LIN {X 0,Y 504.731,Z 518.483,A -85,B 0,C 180,E1 -5683.924,E2 -5683.924} C_VEL
LIN {X 0,Y 504.992,Z 505.216,A -85,B 0,C 180,E1 -5684.251,E2 -5684.251} C_VEL
LIN {X 0,Y 505.338,Z 411.359,A -85,B 0,C 180,E1 -5685.605,E2 -5685.605} C_VEL
LIN {X 0,Y 503.254,Z 400.024,A -85,B 0,C 180,E1 -5685.851,E2 -5685.851} C_VEL
LIN {X 0,Y 503.806,Z 384.288,A -85,B 0,C 180,E1 -5688.925,E2 -5688.925} C_VEL
LIN {X 0,Y 503.812,Z 376.865,A -85,B 0,C 180,E1 -5690.411,E2 -5690.411} C_VEL
LIN {X 0,Y 502.818,Z 371.354,A -85,B 0,C 180,E1 -5691.579,E2 -5691.579} C_VEL
LIN {X 0,Y 502.831,Z 371.357,A -85,B 0,C 180,E1 -5694.791,E2 -5694.791} C_VEL
LIN {X 0,Y 502.836,Z 371.346,A -85,B 0,C 180,E1 -5697.467,E2 -5697.467} C_VEL
LIN {X 0,Y 502.814,Z 371.349,A -85,B 0,C 180,E1 -5700.211,E2 -5700.211} C_VEL
LIN {X 0,Y 502.836,Z 371.349,A -85,B 0,C 180,E1 -5703.031,E2 -5703.031} C_VEL
LIN {X 0,Y 502.778,Z 371.352,A -85,B 0,C 180,E1 -5705.951,E2 -5705.951} C_VEL
LIN {X 0,Y 502.805,Z 371.353,A -85,B 0,C 180,E1 -5708.976,E2 -5708.976} C_VEL
LIN {X 0,Y 502.799,Z 371.352,A -85,B 0,C 180,E1 -5712.14,E2 -5712.14} C_VEL
LIN {X 0,Y 502.806,Z 371.348,A -85,B 0,C 180,E1 -5715.468,E2 -5715.468} C_VEL
LIN {X 0,Y 502.835,Z 371.346,A -85,B 0,C 180,E1 -5717.864,E2 -5717.864} C_VEL
LIN {X 0,Y 502.806,Z 371.35,A -85,B 0,C 180,E1 -5721.024,E2 -5721.024} C_VEL
LIN {X 0,Y 502.78,Z 371.357,A -85,B 0,C 180,E1 -5724.169,E2 -5724.169} C_VEL
LIN {X 0,Y 502.837,Z 371.346,A -85,B 0,C 180,E1 -5726.994,E2 -5726.994} C_VEL
LIN {X 0,Y 502.82,Z 371.352,A -85,B 0,C 180,E1 -5730.065,E2 -5730.065} C_VEL
LIN {X 0,Y 502.839,Z 371.349,A -85,B 0,C 180,E1 -5732.533,E2 -5732.533} C_VEL
LIN {X 0,Y 502.809,Z 371.348,A -85,B 0,C 180,E1 -5735.305,E2 -5735.305} C_VEL
LIN {X 0,Y 502.786,Z 371.354,A -85,B 0,C 180,E1 -5737.827,E2 -5737.827} C_VEL
LIN {X 0,Y 502.831,Z 371.35,A -85,B 0,C 180,E1 -5740.4,E2 -5740.4} C_VEL
LIN {X 0,Y 502.839,Z 371.344,A -85,B 0,C 180,E1 -5742.932,E2 -5742.932} C_VEL
LIN {X 0,Y 502.851,Z 371.344,A -85,B 0,C 180,E1 -5745.429,E2 -5745.429} C_VEL
LIN {X 0,Y 502.883,Z 371.339,A -85,B 0,C 180,E1 -5748.717,E2 -5748.717} C_VEL
LIN {X 0,Y 502.907,Z 371.345,A -85,B 0,C 180,E1 -5751.967,E2 -5751.967} C_VEL
LIN {X 0,Y 502.944,Z 371.334,A -85,B 0,C 180,E1 -5754.387,E2 -5754.387} C_VEL
LIN {X 0,Y 503.03,Z 371.325,A -85,B 0,C 180,E1 -5757.598,E2 -5757.598} C_VEL
LIN {X 0,Y 503.034,Z 371.326,A -85,B 0,C 180,E1 -5760,E2 -5760} C_VEL
LIN {X 0,Y 503.03,Z 371.322,A -85,B 0,C 180,E1 -5762.402,E2 -5762.402} C_VEL
LIN {X 0,Y 502.943,Z 371.338,A -85,B 0,C 180,E1 -5765.613,E2 -5765.613} C_VEL
LIN {X 0,Y 502.886,Z 371.342,A -85,B 0,C 180,E1 -5768.034,E2 -5768.034} C_VEL
LIN {X 0,Y 502.898,Z 371.34,A -85,B 0,C 180,E1 -5771.283,E2 -5771.283} C_VEL
LIN {X 0,Y 502.85,Z 371.343,A -85,B 0,C 180,E1 -5774.571,E2 -5774.571} C_VEL
LIN {X 0,Y 502.861,Z 371.345,A -85,B 0,C 180,E1 -5777.907,E2 -5777.907} C_VEL
LIN {X 0,Y 502.834,Z 371.345,A -85,B 0,C 180,E1 -5780.536,E2 -5780.536} C_VEL
LIN {X 0,Y 502.793,Z 371.353,A -85,B 0,C 180,E1 -5783.041,E2 -5783.041} C_VEL
LIN {X 0,Y 502.826,Z 371.351,A -85,B 0,C 180,E1 -5785.676,E2 -5785.676} C_VEL
LIN {X 0,Y 502.844,Z 371.343,A -85,B 0,C 180,E1 -5788.373,E2 -5788.373} C_VEL
LIN {X 0,Y 502.798,Z 371.356,A -85,B 0,C 180,E1 -5791.499,E2 -5791.499} C_VEL
LIN {X 0,Y 502.793,Z 371.351,A -85,B 0,C 180,E1 -5793.995,E2 -5793.995} C_VEL
LIN {X 0,Y 502.781,Z 371.36,A -85,B 0,C 180,E1 -5797.178,E2 -5797.178} C_VEL
LIN {X 0,Y 502.792,Z 371.35,A -85,B 0,C 180,E1 -5800.015,E2 -5800.015} C_VEL
LIN {X 0,Y 502.807,Z 371.348,A -85,B 0,C 180,E1 -5802.199,E2 -5802.199} C_VEL
LIN {X 0,Y 502.805,Z 371.352,A -85,B 0,C 180,E1 -5805.468,E2 -5805.468} C_VEL
LIN {X 0,Y 502.823,Z 371.353,A -85,B 0,C 180,E1 -5808.934,E2 -5808.934} C_VEL
LIN {X 0,Y 502.797,Z 371.349,A -85,B 0,C 180,E1 -5812.046,E2 -5812.046} C_VEL
LIN {X 0,Y 502.806,Z 371.356,A -85,B 0,C 180,E1 -5815.034,E2 -5815.034} C_VEL
LIN {X 0,Y 502.787,Z 371.351,A -85,B 0,C 180,E1 -5817.915,E2 -5817.915} C_VEL
LIN {X 0,Y 502.828,Z 371.354,A -85,B 0,C 180,E1 -5820.712,E2 -5820.712} C_VEL
LIN {X 0,Y 502.866,Z 371.346,A -85,B 0,C 180,E1 -5823.439,E2 -5823.439} C_VEL
LIN {X 0,Y 502.855,Z 371.502,A -85,B 0,C 180,E1 -5825.552,E2 -5825.552} C_VEL
LIN {X 0,Y 504.53,Z 380.846,A -85,B 0,C 180,E1 -5827.26,E2 -5827.26} C_VEL
LIN {X 0,Y 504.025,Z 395.847,A -85,B 0,C 180,E1 -5829.811,E2 -5829.811} C_VEL
LIN {X 0,Y 503.518,Z 413.319,A -85,B 0,C 180,E1 -5832.746,E2 -5832.746} C_VEL
LIN {X 0,Y 503.256,Z 422.013,A -85,B 0,C 180,E1 -5834.195,E2 -5834.195} C_VEL
LIN {X 0,Y 505.417,Z 435.601,A -85,B 0,C 180,E1 -5834.462,E2 -5834.462} C_VEL
LIN {X 0,Y 504.878,Z 529.981,A -85,B 0,C 180,E1 -5835.823,E2 -5835.823} C_VEL
LIN {X 0,Y 504.597,Z 543.267,A -85,B 0,C 180,E1 -5836.175,E2 -5836.175} C_VEL
LIN {X 0,Y 504.259,Z 556.56,A -85,B 0,C 180,E1 -5836.705,E2 -5836.705} C_VEL
LIN {X 0,Y 503.894,Z 568.939,A -85,B 0,C 180,E1 -5837.389,E2 -5837.389} C_VEL
LIN {X 0,Y 503.606,Z 579.316,A -85,B 0,C 180,E1 -5838.121,E2 -5838.121} C_VEL
LIN {X 0,Y 503.258,Z 589.758,A -85,B 0,C 180,E1 -5839.031,E2 -5839.031} C_VEL
LIN {X 0,Y 502.933,Z 598.295,A -85,B 0,C 180,E1 -5839.94,E2 -5839.94} C_VEL
LIN {X 0,Y 502.66,Z 606.172,A -85,B 0,C 180,E1 -5840.95,E2 -5840.95} C_VEL
LIN {X 0,Y 502.428,Z 613.864,A -85,B 0,C 180,E1 -5842.161,E2 -5842.161} C_VEL
LIN {X 0,Y 502.236,Z 620.547,A -85,B 0,C 180,E1 -5843.482,E2 -5843.482} C_VEL
LIN {X 0,Y 502.182,Z 625.673,A -85,B 0,C 180,E1 -5844.781,E2 -5844.781} C_VEL
LIN {X 0,Y 502.138,Z 629.277,A -85,B 0,C 180,E1 -5845.987,E2 -5845.987} C_VEL
LIN {X 0,Y 502.12,Z 631.136,A -85,B 0,C 180,E1 -5846.79,E2 -5846.79} C_VEL
LIN {X 0,Y 502.091,Z 632.53,A -85,B 0,C 180,E1 -5847.593,E2 -5847.593} C_VEL
LIN {X 0,Y 501.99,Z 634.13,A -85,B 0,C 180,E1 -5849.198,E2 -5849.198} C_VEL
LIN {X 0,Y 501.98,Z 634.346,A -85,B 0,C 180,E1 -5850,E2 -5850} C_VEL
LIN {X 0,Y 502.036,Z 633.525,A -85,B 0,C 180,E1 -5851.604,E2 -5851.604} C_VEL
LIN {X 0,Y 502.091,Z 632.533,A -85,B 0,C 180,E1 -5852.407,E2 -5852.407} C_VEL
LIN {X 0,Y 502.12,Z 631.14,A -85,B 0,C 180,E1 -5853.209,E2 -5853.209} C_VEL
LIN {X 0,Y 502.103,Z 628.209,A -85,B 0,C 180,E1 -5854.415,E2 -5854.415} C_VEL
LIN {X 0,Y 502.235,Z 624.242,A -85,B 0,C 180,E1 -5855.621,E2 -5855.621} C_VEL
LIN {X 0,Y 502.332,Z 618.241,A -85,B 0,C 180,E1 -5857.011,E2 -5857.011} C_VEL
LIN {X 0,Y 502.487,Z 611.47,A -85,B 0,C 180,E1 -5858.242,E2 -5858.242} C_VEL
LIN {X 0,Y 502.74,Z 603.194,A -85,B 0,C 180,E1 -5859.454,E2 -5859.454} C_VEL
LIN {X 0,Y 503.037,Z 594.712,A -85,B 0,C 180,E1 -5860.464,E2 -5860.464} C_VEL
LIN {X 0,Y 503.414,Z 584.231,A -85,B 0,C 180,E1 -5861.475,E2 -5861.475} C_VEL
LIN {X 0,Y 503.713,Z 573.72,A -85,B 0,C 180,E1 -5862.295,E2 -5862.295} C_VEL
LIN {X 0,Y 504.103,Z 562.492,A -85,B 0,C 180,E1 -5862.992,E2 -5862.992} C_VEL
LIN {X 0,Y 504.424,Z 550.833,A -85,B 0,C 180,E1 -5863.547,E2 -5863.547} C_VEL
LIN {X 0,Y 504.721,Z 537.397,A -85,B 0,C 180,E1 -5864.001,E2 -5864.001} C_VEL
LIN {X 0,Y 504.944,Z 524.13,A -85,B 0,C 180,E1 -5864.277,E2 -5864.277} C_VEL
LIN {X 0,Y 505.248,Z 434.384,A -85,B 0,C 180,E1 -5865.561,E2 -5865.561} C_VEL
LIN {X 0,Y 503.306,Z 421.883,A -85,B 0,C 180,E1 -5865.824,E2 -5865.824} C_VEL
LIN {X 0,Y 503.795,Z 403.342,A -85,B 0,C 180,E1 -5868.926,E2 -5868.926} C_VEL
LIN {X 0,Y 504.355,Z 385.848,A -85,B 0,C 180,E1 -5871.885,E2 -5871.885} C_VEL
LIN {X 0,Y 504.419,Z 379.591,A -85,B 0,C 180,E1 -5872.962,E2 -5872.962} C_VEL
LIN {X 0,Y 502.828,Z 371.352,A -85,B 0,C 180,E1 -5874.482,E2 -5874.482} C_VEL
LIN {X 0,Y 502.837,Z 371.352,A -85,B 0,C 180,E1 -5877.467,E2 -5877.467} C_VEL
LIN {X 0,Y 502.812,Z 371.347,A -85,B 0,C 180,E1 -5880.211,E2 -5880.211} C_VEL
LIN {X 0,Y 502.835,Z 371.353,A -85,B 0,C 180,E1 -5883.031,E2 -5883.031} C_VEL
LIN {X 0,Y 502.777,Z 371.352,A -85,B 0,C 180,E1 -5885.951,E2 -5885.951} C_VEL
LIN {X 0,Y 502.805,Z 371.357,A -85,B 0,C 180,E1 -5888.976,E2 -5888.976} C_VEL
LIN {X 0,Y 502.798,Z 371.349,A -85,B 0,C 180,E1 -5892.139,E2 -5892.139} C_VEL
LIN {X 0,Y 502.803,Z 371.35,A -85,B 0,C 180,E1 -5895.468,E2 -5895.468} C_VEL
LIN {X 0,Y 502.832,Z 371.345,A -85,B 0,C 180,E1 -5897.864,E2 -5897.864} C_VEL
LIN {X 0,Y 502.804,Z 371.354,A -85,B 0,C 180,E1 -5901.024,E2 -5901.024} C_VEL
LIN {X 0,Y 502.777,Z 371.353,A -85,B 0,C 180,E1 -5904.169,E2 -5904.169} C_VEL
LIN {X 0,Y 502.835,Z 371.35,A -85,B 0,C 180,E1 -5906.993,E2 -5906.993} C_VEL
LIN {X 0,Y 502.817,Z 371.348,A -85,B 0,C 180,E1 -5910.065,E2 -5910.065} C_VEL
LIN {X 0,Y 502.837,Z 371.352,A -85,B 0,C 180,E1 -5912.533,E2 -5912.533} C_VEL
LIN {X 0,Y 502.806,Z 371.349,A -85,B 0,C 180,E1 -5915.305,E2 -5915.305} C_VEL
LIN {X 0,Y 502.783,Z 371.352,A -85,B 0,C 180,E1 -5917.827,E2 -5917.827} C_VEL
LIN {X 0,Y 502.828,Z 371.353,A -85,B 0,C 180,E1 -5920.4,E2 -5920.4} C_VEL
LIN {X 0,Y 502.833,Z 371.348,A -85,B 0,C 180,E1 -5922.932,E2 -5922.932} C_VEL
LIN {X 0,Y 502.848,Z 371.343,A -85,B 0,C 180,E1 -5925.429,E2 -5925.429} C_VEL
LIN {X 0,Y 502.896,Z 371.341,A -85,B 0,C 180,E1 -5928.717,E2 -5928.717} C_VEL
LIN {X 0,Y 502.884,Z 371.342,A -85,B 0,C 180,E1 -5931.966,E2 -5931.966} C_VEL
LIN {X 0,Y 502.938,Z 371.339,A -85,B 0,C 180,E1 -5934.387,E2 -5934.387} C_VEL
LIN {X 0,Y 503.027,Z 371.322,A -85,B 0,C 180,E1 -5937.598,E2 -5937.598} C_VEL
LIN {X 0,Y 503.031,Z 371.326,A -85,B 0,C 180,E1 -5940,E2 -5940} C_VEL
LIN {X 0,Y 503.028,Z 371.326,A -85,B 0,C 180,E1 -5942.402,E2 -5942.402} C_VEL
LIN {X 0,Y 502.941,Z 371.334,A -85,B 0,C 180,E1 -5945.614,E2 -5945.614} C_VEL
LIN {X 0,Y 502.904,Z 371.344,A -85,B 0,C 180,E1 -5948.033,E2 -5948.033} C_VEL
LIN {X 0,Y 502.881,Z 371.339,A -85,B 0,C 180,E1 -5951.283,E2 -5951.283} C_VEL
LIN {X 0,Y 502.849,Z 371.344,A -85,B 0,C 180,E1 -5954.571,E2 -5954.571} C_VEL
LIN {X 0,Y 502.866,Z 371.349,A -85,B 0,C 180,E1 -5957.907,E2 -5957.907} C_VEL
LIN {X 0,Y 502.832,Z 371.346,A -85,B 0,C 180,E1 -5960.536,E2 -5960.536} C_VEL
LIN {X 0,Y 502.801,Z 371.349,A -85,B 0,C 180,E1 -5963.04,E2 -5963.04} C_VEL
LIN {X 0,Y 502.844,Z 371.35,A -85,B 0,C 180,E1 -5965.676,E2 -5965.676} C_VEL
LIN {X 0,Y 502.844,Z 371.345,A -85,B 0,C 180,E1 -5968.373,E2 -5968.373} C_VEL
LIN {X 0,Y 502.797,Z 371.355,A -85,B 0,C 180,E1 -5971.499,E2 -5971.499} C_VEL
LIN {X 0,Y 502.808,Z 371.348,A -85,B 0,C 180,E1 -5974.444,E2 -5974.444} C_VEL
LIN {X 0,Y 502.784,Z 371.354,A -85,B 0,C 180,E1 -5977.178,E2 -5977.178} C_VEL
LIN {X 0,Y 502.791,Z 371.353,A -85,B 0,C 180,E1 -5980.015,E2 -5980.015} C_VEL
LIN {X 0,Y 502.805,Z 371.349,A -85,B 0,C 180,E1 -5982.199,E2 -5982.199} C_VEL
LIN {X 0,Y 502.804,Z 371.357,A -85,B 0,C 180,E1 -5985.468,E2 -5985.468} C_VEL
LIN {X 0,Y 502.823,Z 371.348,A -85,B 0,C 180,E1 -5988.934,E2 -5988.934} C_VEL
LIN {X 0,Y 502.797,Z 371.35,A -85,B 0,C 180,E1 -5992.046,E2 -5992.046} C_VEL
LIN {X 0,Y 502.813,Z 371.352,A -85,B 0,C 180,E1 -5995.035,E2 -5995.035} C_VEL
LIN {X 0,Y 502.811,Z 371.35,A -85,B 0,C 180,E1 -5997.222,E2 -5997.222} C_VEL
LIN {X 0,Y 502.109,Z 371.438,A -85,B 0,C 180,E1 -5997.891,E2 -5997.891} C_VEL
LIN {X 0,Y 499.244,Z 371.796,A -85,B 0,C 180,E1 -5998.976,E2 -5998.976} C_VEL
LIN {X 0,Y 496.85,Z 372.092,A -85,B 0,C 180,E1 -5999.851,E2 -5999.851} C_VEL
LIN {X 0,Y 495.834,Z 372.217,A -85,B 0,C 180,E1 -6000.527,E2 -6000.527} C_VEL
LIN {X 0,Y 495.756,Z 372.229,A -85,B 0,C 180,E1 -6000.756,E2 -6000.756} C_VEL
LIN {X 0,Y 495.794,Z 372.225,A -85,B 0,C 180,E1 -6003.932,E2 -6003.932} C_VEL
LIN {X 0,Y 495.763,Z 372.234,A -85,B 0,C 180,E1 -6007.139,E2 -6007.139} C_VEL
LIN {X 0,Y 495.813,Z 372.326,A -85,B 0,C 180,E1 -6008.374,E2 -6008.374} C_VEL
LIN {X 0,Y 496.944,Z 379.727,A -85,B 0,C 180,E1 -6009.943,E2 -6009.943} C_VEL
LIN {X 0,Y 496.559,Z 392.479,A -85,B 0,C 180,E1 -6012.497,E2 -6012.497} C_VEL
LIN {X 0,Y 496.313,Z 400.286,A -85,B 0,C 180,E1 -6014.028,E2 -6014.028} C_VEL
LIN {X 0,Y 498.627,Z 413.681,A -85,B 0,C 180,E1 -6014.302,E2 -6014.302} C_VEL
LIN {X 0,Y 498.111,Z 507.421,A -85,B 0,C 180,E1 -6015.679,E2 -6015.679} C_VEL
LIN {X 0,Y 497.803,Z 520.568,A -85,B 0,C 180,E1 -6016.035,E2 -6016.035} C_VEL
LIN {X 0,Y 497.472,Z 532.65,A -85,B 0,C 180,E1 -6016.52,E2 -6016.52} C_VEL
LIN {X 0,Y 497.186,Z 544.94,A -85,B 0,C 180,E1 -6017.195,E2 -6017.195} C_VEL
LIN {X 0,Y 496.796,Z 555.722,A -85,B 0,C 180,E1 -6017.956,E2 -6017.956} C_VEL
LIN {X 0,Y 496.415,Z 566.198,A -85,B 0,C 180,E1 -6018.878,E2 -6018.878} C_VEL
LIN {X 0,Y 496.122,Z 574.758,A -85,B 0,C 180,E1 -6019.801,E2 -6019.801} C_VEL
LIN {X 0,Y 495.779,Z 582.643,A -85,B 0,C 180,E1 -6020.824,E2 -6020.824} C_VEL
LIN {X 0,Y 495.504,Z 590.352,A -85,B 0,C 180,E1 -6022.051,E2 -6022.051} C_VEL
LIN {X 0,Y 495.253,Z 597.424,A -85,B 0,C 180,E1 -6023.482,E2 -6023.482} C_VEL
LIN {X 0,Y 495.128,Z 602.137,A -85,B 0,C 180,E1 -6024.706,E2 -6024.706} C_VEL
LIN {X 0,Y 495.134,Z 605.744,A -85,B 0,C 180,E1 -6025.93,E2 -6025.93} C_VEL
LIN {X 0,Y 495.05,Z 607.611,A -85,B 0,C 180,E1 -6026.745,E2 -6026.745} C_VEL
LIN {X 0,Y 495.025,Z 609.018,A -85,B 0,C 180,E1 -6027.559,E2 -6027.559} C_VEL
LIN {X 0,Y 494.911,Z 610.637,A -85,B 0,C 180,E1 -6029.186,E2 -6029.186} C_VEL
LIN {X 0,Y 494.898,Z 610.874,A -85,B 0,C 180,E1 -6030,E2 -6030} C_VEL
LIN {X 0,Y 494.911,Z 610.689,A -85,B 0,C 180,E1 -6030.814,E2 -6030.814} C_VEL
LIN {X 0,Y 495.025,Z 609.138,A -85,B 0,C 180,E1 -6032.441,E2 -6032.441} C_VEL
LIN {X 0,Y 495.05,Z 607.783,A -85,B 0,C 180,E1 -6033.256,E2 -6033.256} C_VEL
LIN {X 0,Y 495.086,Z 604.918,A -85,B 0,C 180,E1 -6034.478,E2 -6034.478} C_VEL
LIN {X 0,Y 495.236,Z 601.031,A -85,B 0,C 180,E1 -6035.701,E2 -6035.701} C_VEL
LIN {X 0,Y 495.307,Z 596.021,A -85,B 0,C 180,E1 -6036.927,E2 -6036.927} C_VEL
LIN {X 0,Y 495.51,Z 589.71,A -85,B 0,C 180,E1 -6038.154,E2 -6038.154} C_VEL
LIN {X 0,Y 495.771,Z 581.81,A -85,B 0,C 180,E1 -6039.383,E2 -6039.383} C_VEL
LIN {X 0,Y 496.068,Z 573.757,A -85,B 0,C 180,E1 -6040.407,E2 -6040.407} C_VEL
LIN {X 0,Y 496.489,Z 563.927,A -85,B 0,C 180,E1 -6041.431,E2 -6041.431} C_VEL
LIN {X 0,Y 496.886,Z 553.037,A -85,B 0,C 180,E1 -6042.342,E2 -6042.342} C_VEL
LIN {X 0,Y 497.24,Z 542.05,A -85,B 0,C 180,E1 -6043.07,E2 -6043.07} C_VEL
LIN {X 0,Y 497.555,Z 530.092,A -85,B 0,C 180,E1 -6043.686,E2 -6043.686} C_VEL
LIN {X 0,Y 497.89,Z 517.859,A -85,B 0,C 180,E1 -6044.145,E2 -6044.145} C_VEL
LIN {X 0,Y 498.121,Z 505.345,A -85,B 0,C 180,E1 -6044.451,E2 -6044.451} C_VEL
LIN {X 0,Y 498.532,Z 412.239,A -85,B 0,C 180,E1 -6045.812,E2 -6045.812} C_VEL
LIN {X 0,Y 496.306,Z 400.193,A -85,B 0,C 180,E1 -6046.075,E2 -6046.075} C_VEL
LIN {X 0,Y 496.893,Z 383.364,A -85,B 0,C 180,E1 -6049.414,E2 -6049.414} C_VEL
LIN {X 0,Y 496.696,Z 377,A -85,B 0,C 180,E1 -6050.716,E2 -6050.716} C_VEL
LIN {X 0,Y 495.765,Z 372.233,A -85,B 0,C 180,E1 -6051.765,E2 -6051.765} C_VEL
LIN {X 0,Y 495.792,Z 372.232,A -85,B 0,C 180,E1 -6055.167,E2 -6055.167} C_VEL
LIN {X 0,Y 495.784,Z 372.223,A -85,B 0,C 180,E1 -6057.891,E2 -6057.891} C_VEL
LIN {X 0,Y 495.756,Z 372.234,A -85,B 0,C 180,E1 -6060.687,E2 -6060.687} C_VEL
LIN {X 0,Y 495.764,Z 372.226,A -85,B 0,C 180,E1 -6063.564,E2 -6063.564} C_VEL
LIN {X 0,Y 495.732,Z 372.236,A -85,B 0,C 180,E1 -6066.544,E2 -6066.544} C_VEL
LIN {X 0,Y 495.761,Z 372.226,A -85,B 0,C 180,E1 -6069.638,E2 -6069.638} C_VEL
LIN {X 0,Y 495.742,Z 372.236,A -85,B 0,C 180,E1 -6072.507,E2 -6072.507} C_VEL
LIN {X 0,Y 495.754,Z 372.228,A -85,B 0,C 180,E1 -6075.139,E2 -6075.139} C_VEL
LIN {X 0,Y 495.782,Z 372.228,A -85,B 0,C 180,E1 -6078.221,E2 -6078.221} C_VEL
LIN {X 0,Y 495.754,Z 372.227,A -85,B 0,C 180,E1 -6081.408,E2 -6081.408} C_VEL
LIN {X 0,Y 495.753,Z 372.235,A -85,B 0,C 180,E1 -6084.462,E2 -6084.462} C_VEL
LIN {X 0,Y 495.772,Z 372.224,A -85,B 0,C 180,E1 -6087.406,E2 -6087.406} C_VEL
LIN {X 0,Y 495.772,Z 372.233,A -85,B 0,C 180,E1 -6090.254,E2 -6090.254} C_VEL
LIN {X 0,Y 495.829,Z 372.217,A -85,B 0,C 180,E1 -6093.251,E2 -6093.251} C_VEL
LIN {X 0,Y 495.748,Z 372.231,A -85,B 0,C 180,E1 -6096.613,E2 -6096.613} C_VEL
LIN {X 0,Y 495.784,Z 372.223,A -85,B 0,C 180,E1 -6099.324,E2 -6099.324} C_VEL
LIN {X 0,Y 495.804,Z 372.225,A -85,B 0,C 180,E1 -6101.829,E2 -6101.829} C_VEL
LIN {X 0,Y 495.83,Z 372.22,A -85,B 0,C 180,E1 -6104.548,E2 -6104.548} C_VEL
LIN {X 0,Y 495.834,Z 372.225,A -85,B 0,C 180,E1 -6107.965,E2 -6107.965} C_VEL
LIN {X 0,Y 495.845,Z 372.215,A -85,B 0,C 180,E1 -6111.03,E2 -6111.03} C_VEL
LIN {X 0,Y 495.886,Z 372.213,A -85,B 0,C 180,E1 -6113.49,E2 -6113.49} C_VEL
LIN {X 0,Y 495.848,Z 372.215,A -85,B 0,C 180,E1 -6116.75,E2 -6116.75} C_VEL
LIN {X 0,Y 495.876,Z 372.214,A -85,B 0,C 180,E1 -6118.376,E2 -6118.376} C_VEL
LIN {X 0,Y 495.989,Z 372.197,A -85,B 0,C 180,E1 -6120.812,E2 -6120.812} C_VEL
LIN {X 0,Y 495.999,Z 372.197,A -85,B 0,C 180,E1 -6122.436,E2 -6122.436} C_VEL
LIN {X 0,Y 495.901,Z 372.217,A -85,B 0,C 180,E1 -6125.693,E2 -6125.693} C_VEL
LIN {X 0,Y 495.842,Z 372.219,A -85,B 0,C 180,E1 -6128.148,E2 -6128.148} C_VEL
LIN {X 0,Y 495.873,Z 372.218,A -85,B 0,C 180,E1 -6131.445,E2 -6131.445} C_VEL
LIN {X 0,Y 495.796,Z 372.222,A -85,B 0,C 180,E1 -6134.783,E2 -6134.783} C_VEL
LIN {X 0,Y 495.787,Z 372.228,A -85,B 0,C 180,E1 -6137.319,E2 -6137.319} C_VEL
LIN {X 0,Y 495.783,Z 372.227,A -85,B 0,C 180,E1 -6139.89,E2 -6139.89} C_VEL
LIN {X 0,Y 495.764,Z 372.227,A -85,B 0,C 180,E1 -6142.86,E2 -6142.86} C_VEL
LIN {X 0,Y 495.785,Z 372.224,A -85,B 0,C 180,E1 -6146.068,E2 -6146.068} C_VEL
LIN {X 0,Y 495.776,Z 372.226,A -85,B 0,C 180,E1 -6148.815,E2 -6148.815} C_VEL
LIN {X 0,Y 495.76,Z 372.229,A -85,B 0,C 180,E1 -6151.725,E2 -6151.725} C_VEL
LIN {X 0,Y 495.766,Z 372.227,A -85,B 0,C 180,E1 -6154.693,E2 -6154.693} C_VEL
LIN {X 0,Y 495.733,Z 372.233,A -85,B 0,C 180,E1 -6157.561,E2 -6157.561} C_VEL
LIN {X 0,Y 495.77,Z 372.227,A -85,B 0,C 180,E1 -6160.7,E2 -6160.7} C_VEL
LIN {X 0,Y 495.738,Z 372.229,A -85,B 0,C 180,E1 -6164.001,E2 -6164.001} C_VEL
LIN {X 0,Y 495.729,Z 372.238,A -85,B 0,C 180,E1 -6167.117,E2 -6167.117} C_VEL
LIN {X 0,Y 495.763,Z 372.226,A -85,B 0,C 180,E1 -6169.953,E2 -6169.953} C_VEL
LIN {X 0,Y 495.732,Z 372.232,A -85,B 0,C 180,E1 -6172.553,E2 -6172.553} C_VEL
LIN {X 0,Y 495.785,Z 372.225,A -85,B 0,C 180,E1 -6175.457,E2 -6175.457} C_VEL
LIN {X 0,Y 495.759,Z 372.228,A -85,B 0,C 180,E1 -6178.364,E2 -6178.364} C_VEL
LIN {X 0,Y 495.791,Z 372.226,A -85,B 0,C 180,E1 -6181.507,E2 -6181.507} C_VEL
LIN {X 0,Y 495.795,Z 372.226,A -85,B 0,C 180,E1 -6183.932,E2 -6183.932} C_VEL
LIN {X 0,Y 495.834,Z 372.431,A -85,B 0,C 180,E1 -6185.373,E2 -6185.373} C_VEL
LIN {X 0,Y 497.564,Z 381.957,A -85,B 0,C 180,E1 -6187.143,E2 -6187.143} C_VEL
LIN {X 0,Y 497.058,Z 396.952,A -85,B 0,C 180,E1 -6189.732,E2 -6189.732} C_VEL
LIN {X 0,Y 496.496,Z 414.411,A -85,B 0,C 180,E1 -6192.707,E2 -6192.707} C_VEL
LIN {X 0,Y 496.261,Z 421.833,A -85,B 0,C 180,E1 -6193.965,E2 -6193.965} C_VEL
LIN {X 0,Y 498.6,Z 436.905,A -85,B 0,C 180,E1 -6194.265,E2 -6194.265} C_VEL
LIN {X 0,Y 498.007,Z 529.814,A -85,B 0,C 180,E1 -6195.624,E2 -6195.624} C_VEL
LIN {X 0,Y 497.718,Z 543.1,A -85,B 0,C 180,E1 -6195.98,E2 -6195.98} C_VEL
LIN {X 0,Y 497.368,Z 555.27,A -85,B 0,C 180,E1 -6196.465,E2 -6196.465} C_VEL
LIN {X 0,Y 497.02,Z 567.616,A -85,B 0,C 180,E1 -6197.136,E2 -6197.136} C_VEL
LIN {X 0,Y 496.654,Z 577.853,A -85,B 0,C 180,E1 -6197.849,E2 -6197.849} C_VEL
LIN {X 0,Y 496.304,Z 588.518,A -85,B 0,C 180,E1 -6198.772,E2 -6198.772} C_VEL
LIN {X 0,Y 495.89,Z 598.126,A -85,B 0,C 180,E1 -6199.796,E2 -6199.796} C_VEL
LIN {X 0,Y 495.62,Z 606.004,A -85,B 0,C 180,E1 -6200.82,E2 -6200.82} C_VEL
LIN {X 0,Y 495.37,Z 613.696,A -85,B 0,C 180,E1 -6202.049,E2 -6202.049} C_VEL
LIN {X 0,Y 495.164,Z 620.787,A -85,B 0,C 180,E1 -6203.48,E2 -6203.48} C_VEL
LIN {X 0,Y 495.116,Z 625.506,A -85,B 0,C 180,E1 -6204.706,E2 -6204.706} C_VEL
LIN {X 0,Y 495.032,Z 629.109,A -85,B 0,C 180,E1 -6205.929,E2 -6205.929} C_VEL
LIN {X 0,Y 495.042,Z 630.969,A -85,B 0,C 180,E1 -6206.744,E2 -6206.744} C_VEL
LIN {X 0,Y 494.998,Z 632.362,A -85,B 0,C 180,E1 -6207.559,E2 -6207.559} C_VEL
LIN {X 0,Y 494.962,Z 633.357,A -85,B 0,C 180,E1 -6208.373,E2 -6208.373} C_VEL
LIN {X 0,Y 494.898,Z 634.179,A -85,B 0,C 180,E1 -6210,E2 -6210} C_VEL
LIN {X 0,Y 494.962,Z 633.359,A -85,B 0,C 180,E1 -6211.627,E2 -6211.627} C_VEL
LIN {X 0,Y 494.998,Z 632.366,A -85,B 0,C 180,E1 -6212.441,E2 -6212.441} C_VEL
LIN {X 0,Y 495.042,Z 630.973,A -85,B 0,C 180,E1 -6213.255,E2 -6213.255} C_VEL
LIN {X 0,Y 495.009,Z 628.041,A -85,B 0,C 180,E1 -6214.479,E2 -6214.479} C_VEL
LIN {X 0,Y 495.151,Z 624.075,A -85,B 0,C 180,E1 -6215.702,E2 -6215.702} C_VEL
LIN {X 0,Y 495.257,Z 617.972,A -85,B 0,C 180,E1 -6217.133,E2 -6217.133} C_VEL
LIN {X 0,Y 495.432,Z 611.302,A -85,B 0,C 180,E1 -6218.36,E2 -6218.36} C_VEL
LIN {X 0,Y 495.714,Z 603.026,A -85,B 0,C 180,E1 -6219.589,E2 -6219.589} C_VEL
LIN {X 0,Y 496.025,Z 594.544,A -85,B 0,C 180,E1 -6220.614,E2 -6220.614} C_VEL
LIN {X 0,Y 496.452,Z 584.063,A -85,B 0,C 180,E1 -6221.638,E2 -6221.638} C_VEL
LIN {X 0,Y 496.777,Z 572.636,A -85,B 0,C 180,E1 -6222.536,E2 -6222.536} C_VEL
LIN {X 0,Y 497.194,Z 560.402,A -85,B 0,C 180,E1 -6223.279,E2 -6223.279} C_VEL
LIN {X 0,Y 497.562,Z 548.061,A -85,B 0,C 180,E1 -6223.842,E2 -6223.842} C_VEL
LIN {X 0,Y 497.888,Z 535.4,A -85,B 0,C 180,E1 -6224.249,E2 -6224.249} C_VEL
LIN {X 0,Y 498.111,Z 522.188,A -85,B 0,C 180,E1 -6224.503,E2 -6224.503} C_VEL
LIN {X 0,Y 498.419,Z 435.006,A -85,B 0,C 180,E1 -6225.768,E2 -6225.768} C_VEL
LIN {X 0,Y 496.283,Z 421.809,A -85,B 0,C 180,E1 -6226.037,E2 -6226.037} C_VEL
LIN {X 0,Y 496.805,Z 404.441,A -85,B 0,C 180,E1 -6228.988,E2 -6228.988} C_VEL
LIN {X 0,Y 497.402,Z 386.955,A -85,B 0,C 180,E1 -6231.989,E2 -6231.989} C_VEL
LIN {X 0,Y 497.576,Z 381.955,A -85,B 0,C 180,E1 -6232.856,E2 -6232.856} C_VEL
LIN {X 0,Y 495.808,Z 372.227,A -85,B 0,C 180,E1 -6234.668,E2 -6234.668} C_VEL
LIN {X 0,Y 495.816,Z 372.226,A -85,B 0,C 180,E1 -6236.974,E2 -6236.974} C_VEL
LIN {X 0,Y 495.768,Z 372.225,A -85,B 0,C 180,E1 -6240.147,E2 -6240.147} C_VEL
LIN {X 0,Y 495.796,Z 372.228,A -85,B 0,C 180,E1 -6243.245,E2 -6243.245} C_VEL
LIN {X 0,Y 495.723,Z 372.231,A -85,B 0,C 180,E1 -6246.089,E2 -6246.089} C_VEL
LIN {X 0,Y 495.767,Z 372.23,A -85,B 0,C 180,E1 -6248.768,E2 -6248.768} C_VEL
LIN {X 0,Y 495.759,Z 372.226,A -85,B 0,C 180,E1 -6251.781,E2 -6251.781} C_VEL
LIN {X 0,Y 495.752,Z 372.232,A -85,B 0,C 180,E1 -6255.139,E2 -6255.139} C_VEL
LIN {X 0,Y 495.78,Z 372.225,A -85,B 0,C 180,E1 -6258.221,E2 -6258.221} C_VEL
LIN {X 0,Y 495.752,Z 372.228,A -85,B 0,C 180,E1 -6261.408,E2 -6261.408} C_VEL
LIN {X 0,Y 495.75,Z 372.232,A -85,B 0,C 180,E1 -6264.462,E2 -6264.462} C_VEL
LIN {X 0,Y 495.77,Z 372.226,A -85,B 0,C 180,E1 -6267.406,E2 -6267.406} C_VEL
LIN {X 0,Y 495.769,Z 372.228,A -85,B 0,C 180,E1 -6270.254,E2 -6270.254} C_VEL
LIN {X 0,Y 495.826,Z 372.219,A -85,B 0,C 180,E1 -6273.251,E2 -6273.251} C_VEL
LIN {X 0,Y 495.746,Z 372.236,A -85,B 0,C 180,E1 -6276.613,E2 -6276.613} C_VEL
LIN {X 0,Y 495.781,Z 372.224,A -85,B 0,C 180,E1 -6279.324,E2 -6279.324} C_VEL
LIN {X 0,Y 495.796,Z 372.223,A -85,B 0,C 180,E1 -6281.829,E2 -6281.829} C_VEL
LIN {X 0,Y 495.827,Z 372.225,A -85,B 0,C 180,E1 -6284.548,E2 -6284.548} C_VEL
LIN {X 0,Y 495.88,Z 372.214,A -85,B 0,C 180,E1 -6287.939,E2 -6287.939} C_VEL
LIN {X 0,Y 495.84,Z 372.217,A -85,B 0,C 180,E1 -6291.03,E2 -6291.03} C_VEL
LIN {X 0,Y 495.868,Z 372.213,A -85,B 0,C 180,E1 -6293.49,E2 -6293.49} C_VEL
LIN {X 0,Y 495.845,Z 372.218,A -85,B 0,C 180,E1 -6296.75,E2 -6296.75} C_VEL
LIN {X 0,Y 495.874,Z 372.219,A -85,B 0,C 180,E1 -6298.376,E2 -6298.376} C_VEL
LIN {X 0,Y 496.008,Z 372.196,A -85,B 0,C 180,E1 -6300.812,E2 -6300.812} C_VEL
LIN {X 0,Y 495.846,Z 372.215,A -85,B 0,C 180,E1 -6303.25,E2 -6303.25} C_VEL
LIN {X 0,Y 495.883,Z 372.214,A -85,B 0,C 180,E1 -6306.51,E2 -6306.51} C_VEL
LIN {X 0,Y 495.842,Z 372.216,A -85,B 0,C 180,E1 -6308.97,E2 -6308.97} C_VEL
LIN {X 0,Y 495.832,Z 372.226,A -85,B 0,C 180,E1 -6312.035,E2 -6312.035} C_VEL
LIN {X 0,Y 495.827,Z 372.22,A -85,B 0,C 180,E1 -6315.452,E2 -6315.452} C_VEL
LIN {X 0,Y 495.81,Z 372.224,A -85,B 0,C 180,E1 -6318.247,E2 -6318.247} C_VEL
LIN {X 0,Y 495.777,Z 372.224,A -85,B 0,C 180,E1 -6320.756,E2 -6320.756} C_VEL
LIN {X 0,Y 495.757,Z 372.229,A -85,B 0,C 180,E1 -6323.387,E2 -6323.387} C_VEL
LIN {X 0,Y 495.794,Z 372.227,A -85,B 0,C 180,E1 -6326.068,E2 -6326.068} C_VEL
LIN {X 0,Y 495.775,Z 372.224,A -85,B 0,C 180,E1 -6328.815,E2 -6328.815} C_VEL
LIN {X 0,Y 495.76,Z 372.235,A -85,B 0,C 180,E1 -6331.726,E2 -6331.726} C_VEL
LIN {X 0,Y 495.778,Z 372.224,A -85,B 0,C 180,E1 -6334.695,E2 -6334.695} C_VEL
LIN {X 0,Y 495.735,Z 372.237,A -85,B 0,C 180,E1 -6337.561,E2 -6337.561} C_VEL
LIN {X 0,Y 495.769,Z 372.225,A -85,B 0,C 180,E1 -6340.7,E2 -6340.7} C_VEL
LIN {X 0,Y 495.738,Z 372.235,A -85,B 0,C 180,E1 -6343.696,E2 -6343.696} C_VEL
LIN {X 0,Y 495.732,Z 372.23,A -85,B 0,C 180,E1 -6346.305,E2 -6346.305} C_VEL
LIN {X 0,Y 495.769,Z 372.231,A -85,B 0,C 180,E1 -6349.3,E2 -6349.3} C_VEL
LIN {X 0,Y 495.734,Z 372.229,A -85,B 0,C 180,E1 -6352.439,E2 -6352.439} C_VEL
LIN {X 0,Y 495.789,Z 372.23,A -85,B 0,C 180,E1 -6355.458,E2 -6355.458} C_VEL
LIN {X 0,Y 495.758,Z 372.226,A -85,B 0,C 180,E1 -6358.364,E2 -6358.364} C_VEL
LIN {X 0,Y 495.756,Z 372.229,A -85,B 0,C 180,E1 -6360.756,E2 -6360.756} C_VEL
LIN {X 0,Y 495.099,Z 372.316,A -85,B 0,C 180,E1 -6361.435,E2 -6361.435} C_VEL
LIN {X 0,Y 492.243,Z 372.67,A -85,B 0,C 180,E1 -6362.537,E2 -6362.537} C_VEL
LIN {X 0,Y 489.834,Z 372.971,A -85,B 0,C 180,E1 -6363.426,E2 -6363.426} C_VEL
LIN {X 0,Y 488.818,Z 373.094,A -85,B 0,C 180,E1 -6364.112,E2 -6364.112} C_VEL
LIN {X 0,Y 488.745,Z 373.103,A -85,B 0,C 180,E1 -6364.345,E2 -6364.345} C_VEL
LIN {X 0,Y 488.726,Z 373.111,A -85,B 0,C 180,E1 -6367.153,E2 -6367.153} C_VEL
LIN {X 0,Y 488.759,Z 373.259,A -85,B 0,C 180,E1 -6368.213,E2 -6368.213} C_VEL
LIN {X 0,Y 489.991,Z 380.927,A -85,B 0,C 180,E1 -6369.865,E2 -6369.865} C_VEL
LIN {X 0,Y 489.579,Z 393.693,A -85,B 0,C 180,E1 -6372.455,E2 -6372.455} C_VEL
LIN {X 0,Y 489.357,Z 400.405,A -85,B 0,C 180,E1 -6373.789,E2 -6373.789} C_VEL
LIN {X 0,Y 491.809,Z 414.288,A -85,B 0,C 180,E1 -6374.085,E2 -6374.085} C_VEL
LIN {X 0,Y 491.239,Z 507.614,A -85,B 0,C 180,E1 -6375.474,E2 -6375.474} C_VEL
LIN {X 0,Y 490.917,Z 520.752,A -85,B 0,C 180,E1 -6375.835,E2 -6375.835} C_VEL
LIN {X 0,Y 490.578,Z 532.83,A -85,B 0,C 180,E1 -6376.327,E2 -6376.327} C_VEL
LIN {X 0,Y 490.291,Z 543.746,A -85,B 0,C 180,E1 -6376.923,E2 -6376.923} C_VEL
LIN {X 0,Y 489.922,Z 554.609,A -85,B 0,C 180,E1 -6377.679,E2 -6377.679} C_VEL
LIN {X 0,Y 489.465,Z 565.307,A -85,B 0,C 180,E1 -6378.613,E2 -6378.613} C_VEL
LIN {X 0,Y 489.138,Z 574.93,A -85,B 0,C 180,E1 -6379.654,E2 -6379.654} C_VEL
LIN {X 0,Y 488.743,Z 582.816,A -85,B 0,C 180,E1 -6380.69,E2 -6380.69} C_VEL
LIN {X 0,Y 488.46,Z 590.523,A -85,B 0,C 180,E1 -6381.936,E2 -6381.936} C_VEL
LIN {X 0,Y 488.183,Z 597.595,A -85,B 0,C 180,E1 -6383.387,E2 -6383.387} C_VEL
LIN {X 0,Y 488.074,Z 602.306,A -85,B 0,C 180,E1 -6384.63,E2 -6384.63} C_VEL
LIN {X 0,Y 488.036,Z 605.913,A -85,B 0,C 180,E1 -6385.871,E2 -6385.871} C_VEL
LIN {X 0,Y 487.977,Z 607.779,A -85,B 0,C 180,E1 -6386.698,E2 -6386.698} C_VEL
LIN {X 0,Y 487.933,Z 609.186,A -85,B 0,C 180,E1 -6387.524,E2 -6387.524} C_VEL
LIN {X 0,Y 487.834,Z 610.804,A -85,B 0,C 180,E1 -6389.175,E2 -6389.175} C_VEL
LIN {X 0,Y 487.819,Z 611.041,A -85,B 0,C 180,E1 -6390,E2 -6390} C_VEL
LIN {X 0,Y 487.834,Z 610.855,A -85,B 0,C 180,E1 -6390.826,E2 -6390.826} C_VEL
LIN {X 0,Y 487.934,Z 609.305,A -85,B 0,C 180,E1 -6392.477,E2 -6392.477} C_VEL
LIN {X 0,Y 487.978,Z 607.949,A -85,B 0,C 180,E1 -6393.303,E2 -6393.303} C_VEL
LIN {X 0,Y 487.987,Z 605.084,A -85,B 0,C 180,E1 -6394.543,E2 -6394.543} C_VEL
LIN {X 0,Y 488.188,Z 600.152,A -85,B 0,C 180,E1 -6396.066,E2 -6396.066} C_VEL
LIN {X 0,Y 488.293,Z 594.212,A -85,B 0,C 180,E1 -6397.443,E2 -6397.443} C_VEL
LIN {X 0,Y 488.572,Z 587.424,A -85,B 0,C 180,E1 -6398.687,E2 -6398.687} C_VEL
LIN {X 0,Y 488.89,Z 578.949,A -85,B 0,C 180,E1 -6399.934,E2 -6399.934} C_VEL
LIN {X 0,Y 489.287,Z 570.229,A -85,B 0,C 180,E1 -6400.972,E2 -6400.972} C_VEL
LIN {X 0,Y 489.717,Z 559.49,A -85,B 0,C 180,E1 -6402.011,E2 -6402.011} C_VEL
LIN {X 0,Y 490.073,Z 549.442,A -85,B 0,C 180,E1 -6402.794,E2 -6402.794} C_VEL
LIN {X 0,Y 490.448,Z 538.625,A -85,B 0,C 180,E1 -6403.466,E2 -6403.466} C_VEL
LIN {X 0,Y 490.773,Z 526.588,A -85,B 0,C 180,E1 -6404.037,E2 -6404.037} C_VEL
LIN {X 0,Y 491.079,Z 513.482,A -85,B 0,C 180,E1 -6404.478,E2 -6404.478} C_VEL
LIN {X 0,Y 491.287,Z 500.883,A -85,B 0,C 180,E1 -6404.736,E2 -6404.736} C_VEL
LIN {X 0,Y 491.73,Z 413.091,A -85,B 0,C 180,E1 -6406.026,E2 -6406.026} C_VEL
LIN {X 0,Y 489.331,Z 400.363,A -85,B 0,C 180,E1 -6406.307,E2 -6406.307} C_VEL
LIN {X 0,Y 489.946,Z 384.562,A -85,B 0,C 180,E1 -6409.482,E2 -6409.482} C_VEL
LIN {X 0,Y 489.869,Z 379.254,A -85,B 0,C 180,E1 -6410.579,E2 -6410.579} C_VEL
LIN {X 0,Y 488.729,Z 373.109,A -85,B 0,C 180,E1 -6411.956,E2 -6411.956} C_VEL
LIN {X 0,Y 488.751,Z 373.106,A -85,B 0,C 180,E1 -6415.556,E2 -6415.556} C_VEL
LIN {X 0,Y 488.748,Z 373.102,A -85,B 0,C 180,E1 -6418.329,E2 -6418.329} C_VEL
LIN {X 0,Y 488.696,Z 373.109,A -85,B 0,C 180,E1 -6421.18,E2 -6421.18} C_VEL
LIN {X 0,Y 488.736,Z 373.102,A -85,B 0,C 180,E1 -6424.113,E2 -6424.113} C_VEL
LIN {X 0,Y 488.683,Z 373.11,A -85,B 0,C 180,E1 -6427.159,E2 -6427.159} C_VEL
LIN {X 0,Y 488.722,Z 373.107,A -85,B 0,C 180,E1 -6430.345,E2 -6430.345} C_VEL
LIN {X 0,Y 488.691,Z 373.107,A -85,B 0,C 180,E1 -6433.655,E2 -6433.655} C_VEL
LIN {X 0,Y 488.698,Z 373.112,A -85,B 0,C 180,E1 -6436.347,E2 -6436.347} C_VEL
LIN {X 0,Y 488.724,Z 373.11,A -85,B 0,C 180,E1 -6438.586,E2 -6438.586} C_VEL
LIN {X 0,Y 488.684,Z 373.109,A -85,B 0,C 180,E1 -6441.8,E2 -6441.8} C_VEL
LIN {X 0,Y 488.728,Z 373.103,A -85,B 0,C 180,E1 -6445.053,E2 -6445.053} C_VEL
LIN {X 0,Y 488.709,Z 373.109,A -85,B 0,C 180,E1 -6448.046,E2 -6448.046} C_VEL
LIN {X 0,Y 488.729,Z 373.105,A -85,B 0,C 180,E1 -6450.73,E2 -6450.73} C_VEL
LIN {X 0,Y 488.758,Z 373.099,A -85,B 0,C 180,E1 -6453.528,E2 -6453.528} C_VEL
LIN {X 0,Y 488.686,Z 373.116,A -85,B 0,C 180,E1 -6456.254,E2 -6456.254} C_VEL
LIN {X 0,Y 488.752,Z 373.099,A -85,B 0,C 180,E1 -6459.176,E2 -6459.176} C_VEL
LIN {X 0,Y 488.765,Z 373.1,A -85,B 0,C 180,E1 -6461.628,E2 -6461.628} C_VEL
LIN {X 0,Y 488.768,Z 373.097,A -85,B 0,C 180,E1 -6465,E2 -6465} C_VEL
LIN {X 0,Y 488.812,Z 373.095,A -85,B 0,C 180,E1 -6468.388,E2 -6468.388} C_VEL
LIN {X 0,Y 488.822,Z 373.096,A -85,B 0,C 180,E1 -6471.734,E2 -6471.734} C_VEL
LIN {X 0,Y 488.861,Z 373.09,A -85,B 0,C 180,E1 -6474.224,E2 -6474.224} C_VEL
LIN {X 0,Y 488.967,Z 373.076,A -85,B 0,C 180,E1 -6477.529,E2 -6477.529} C_VEL
LIN {X 0,Y 488.94,Z 373.076,A -85,B 0,C 180,E1 -6480.824,E2 -6480.824} C_VEL
LIN {X 0,Y 488.967,Z 373.073,A -85,B 0,C 180,E1 -6482.471,E2 -6482.471} C_VEL
LIN {X 0,Y 488.861,Z 373.094,A -85,B 0,C 180,E1 -6485.776,E2 -6485.776} C_VEL
LIN {X 0,Y 488.79,Z 373.096,A -85,B 0,C 180,E1 -6488.267,E2 -6488.267} C_VEL
LIN {X 0,Y 488.835,Z 373.097,A -85,B 0,C 180,E1 -6491.612,E2 -6491.612} C_VEL
LIN {X 0,Y 488.768,Z 373.099,A -85,B 0,C 180,E1 -6495,E2 -6495} C_VEL
LIN {X 0,Y 488.76,Z 373.098,A -85,B 0,C 180,E1 -6498.442,E2 -6498.442} C_VEL
LIN {X 0,Y 488.712,Z 373.107,A -85,B 0,C 180,E1 -6501.071,E2 -6501.071} C_VEL
LIN {X 0,Y 488.685,Z 373.112,A -85,B 0,C 180,E1 -6503.746,E2 -6503.746} C_VEL
LIN {X 0,Y 488.796,Z 373.096,A -85,B 0,C 180,E1 -6506.943,E2 -6506.943} C_VEL
LIN {X 0,Y 488.714,Z 373.104,A -85,B 0,C 180,E1 -6510.363,E2 -6510.363} C_VEL
LIN {X 0,Y 488.733,Z 373.107,A -85,B 0,C 180,E1 -6513.483,E2 -6513.483} C_VEL
LIN {X 0,Y 488.686,Z 373.107,A -85,B 0,C 180,E1 -6516.354,E2 -6516.354} C_VEL
LIN {X 0,Y 488.705,Z 373.113,A -85,B 0,C 180,E1 -6519.254,E2 -6519.254} C_VEL
LIN {X 0,Y 488.711,Z 373.107,A -85,B 0,C 180,E1 -6521.6,E2 -6521.6} C_VEL
LIN {X 0,Y 488.716,Z 373.108,A -85,B 0,C 180,E1 -6524.801,E2 -6524.801} C_VEL
LIN {X 0,Y 488.695,Z 373.109,A -85,B 0,C 180,E1 -6527.474,E2 -6527.474} C_VEL
LIN {X 0,Y 488.737,Z 373.102,A -85,B 0,C 180,E1 -6529.676,E2 -6529.676} C_VEL
LIN {X 0,Y 488.684,Z 373.114,A -85,B 0,C 180,E1 -6532.841,E2 -6532.841} C_VEL
LIN {X 0,Y 488.736,Z 373.101,A -85,B 0,C 180,E1 -6535.887,E2 -6535.887} C_VEL
LIN {X 0,Y 488.696,Z 373.114,A -85,B 0,C 180,E1 -6538.82,E2 -6538.82} C_VEL
LIN {X 0,Y 488.748,Z 373.103,A -85,B 0,C 180,E1 -6541.671,E2 -6541.671} C_VEL
LIN {X 0,Y 488.751,Z 373.105,A -85,B 0,C 180,E1 -6544.444,E2 -6544.444} C_VEL
LIN {X 0,Y 488.768,Z 373.168,A -85,B 0,C 180,E1 -6545.151,E2 -6545.151} C_VEL
LIN {X 0,Y 490.537,Z 382.485,A -85,B 0,C 180,E1 -6546.916,E2 -6546.916} C_VEL
LIN {X 0,Y 490.383,Z 391.51,A -85,B 0,C 180,E1 -6548.511,E2 -6548.511} C_VEL
LIN {X 0,Y 489.649,Z 411.77,A -85,B 0,C 180,E1 -6552.025,E2 -6552.025} C_VEL
LIN {X 0,Y 489.298,Z 421.808,A -85,B 0,C 180,E1 -6553.736,E2 -6553.736} C_VEL
LIN {X 0,Y 491.747,Z 437.03,A -85,B 0,C 180,E1 -6554.045,E2 -6554.045} C_VEL
LIN {X 0,Y 491.143,Z 529.649,A -85,B 0,C 180,E1 -6555.418,E2 -6555.418} C_VEL
LIN {X 0,Y 490.847,Z 542.934,A -85,B 0,C 180,E1 -6555.78,E2 -6555.78} C_VEL
LIN {X 0,Y 490.456,Z 555.103,A -85,B 0,C 180,E1 -6556.271,E2 -6556.271} C_VEL
LIN {X 0,Y 490.077,Z 567.384,A -85,B 0,C 180,E1 -6556.946,E2 -6556.946} C_VEL
LIN {X 0,Y 489.692,Z 577.685,A -85,B 0,C 180,E1 -6557.673,E2 -6557.673} C_VEL
LIN {X 0,Y 489.313,Z 588.351,A -85,B 0,C 180,E1 -6558.609,E2 -6558.609} C_VEL
LIN {X 0,Y 488.874,Z 597.959,A -85,B 0,C 180,E1 -6559.648,E2 -6559.648} C_VEL
LIN {X 0,Y 488.568,Z 605.836,A -85,B 0,C 180,E1 -6560.687,E2 -6560.687} C_VEL
LIN {X 0,Y 488.322,Z 613.529,A -85,B 0,C 180,E1 -6561.933,E2 -6561.933} C_VEL
LIN {X 0,Y 488.101,Z 620.62,A -85,B 0,C 180,E1 -6563.385,E2 -6563.385} C_VEL
LIN {X 0,Y 488.03,Z 625.338,A -85,B 0,C 180,E1 -6564.629,E2 -6564.629} C_VEL
LIN {X 0,Y 487.928,Z 628.942,A -85,B 0,C 180,E1 -6565.87,E2 -6565.87} C_VEL
LIN {X 0,Y 487.964,Z 630.802,A -85,B 0,C 180,E1 -6566.697,E2 -6566.697} C_VEL
LIN {X 0,Y 487.891,Z 633.19,A -85,B 0,C 180,E1 -6568.349,E2 -6568.349} C_VEL
LIN {X 0,Y 487.819,Z 634.012,A -85,B 0,C 180,E1 -6570,E2 -6570} C_VEL
LIN {X 0,Y 487.891,Z 633.192,A -85,B 0,C 180,E1 -6571.651,E2 -6571.651} C_VEL
LIN {X 0,Y 487.964,Z 630.807,A -85,B 0,C 180,E1 -6573.303,E2 -6573.303} C_VEL
LIN {X 0,Y 487.922,Z 627.874,A -85,B 0,C 180,E1 -6574.544,E2 -6574.544} C_VEL
LIN {X 0,Y 488.068,Z 623.907,A -85,B 0,C 180,E1 -6575.785,E2 -6575.785} C_VEL
LIN {X 0,Y 488.183,Z 617.804,A -85,B 0,C 180,E1 -6577.236,E2 -6577.236} C_VEL
LIN {X 0,Y 488.368,Z 611.134,A -85,B 0,C 180,E1 -6578.482,E2 -6578.482} C_VEL
LIN {X 0,Y 488.687,Z 602.858,A -85,B 0,C 180,E1 -6579.729,E2 -6579.729} C_VEL
LIN {X 0,Y 489.026,Z 594.377,A -85,B 0,C 180,E1 -6580.768,E2 -6580.768} C_VEL
LIN {X 0,Y 489.492,Z 583.896,A -85,B 0,C 180,E1 -6581.806,E2 -6581.806} C_VEL
LIN {X 0,Y 489.832,Z 572.617,A -85,B 0,C 180,E1 -6582.706,E2 -6582.706} C_VEL
LIN {X 0,Y 490.221,Z 562.156,A -85,B 0,C 180,E1 -6583.366,E2 -6583.366} C_VEL
LIN {X 0,Y 490.592,Z 550.497,A -85,B 0,C 180,E1 -6583.937,E2 -6583.937} C_VEL
LIN {X 0,Y 490.977,Z 537.062,A -85,B 0,C 180,E1 -6584.401,E2 -6584.401} C_VEL
LIN {X 0,Y 491.215,Z 523.793,A -85,B 0,C 180,E1 -6584.685,E2 -6584.685} C_VEL
LIN {X 0,Y 491.617,Z 436.069,A -85,B 0,C 180,E1 -6585.974,E2 -6585.974} C_VEL
LIN {X 0,Y 489.324,Z 421.562,A -85,B 0,C 180,E1 -6586.286,E2 -6586.286} C_VEL
LIN {X 0,Y 489.865,Z 404.29,A -85,B 0,C 180,E1 -6589.267,E2 -6589.267} C_VEL
LIN {X 0,Y 490.631,Z 385.565,A -85,B 0,C 180,E1 -6592.531,E2 -6592.531} C_VEL
LIN {X 0,Y 490.229,Z 380.6,A -85,B 0,C 180,E1 -6593.434,E2 -6593.434} C_VEL
LIN {X 0,Y 488.75,Z 373.106,A -85,B 0,C 180,E1 -6594.878,E2 -6594.878} C_VEL
LIN {X 0,Y 488.749,Z 373.108,A -85,B 0,C 180,E1 -6597.397,E2 -6597.397} C_VEL
LIN {X 0,Y 488.713,Z 373.104,A -85,B 0,C 180,E1 -6600.363,E2 -6600.363} C_VEL
LIN {X 0,Y 488.738,Z 373.104,A -85,B 0,C 180,E1 -6603.484,E2 -6603.484} C_VEL
LIN {X 0,Y 488.685,Z 373.108,A -85,B 0,C 180,E1 -6606.355,E2 -6606.355} C_VEL
LIN {X 0,Y 488.704,Z 373.11,A -85,B 0,C 180,E1 -6609.254,E2 -6609.254} C_VEL
LIN {X 0,Y 488.71,Z 373.105,A -85,B 0,C 180,E1 -6611.6,E2 -6611.6} C_VEL
LIN {X 0,Y 488.714,Z 373.111,A -85,B 0,C 180,E1 -6614.801,E2 -6614.801} C_VEL
LIN {X 0,Y 488.698,Z 373.107,A -85,B 0,C 180,E1 -6617.475,E2 -6617.475} C_VEL
LIN {X 0,Y 488.735,Z 373.101,A -85,B 0,C 180,E1 -6619.677,E2 -6619.677} C_VEL
LIN {X 0,Y 488.681,Z 373.116,A -85,B 0,C 180,E1 -6622.841,E2 -6622.841} C_VEL
LIN {X 0,Y 488.733,Z 373.102,A -85,B 0,C 180,E1 -6625.887,E2 -6625.887} C_VEL
LIN {X 0,Y 488.695,Z 373.113,A -85,B 0,C 180,E1 -6628.82,E2 -6628.82} C_VEL
LIN {X 0,Y 488.747,Z 373.1,A -85,B 0,C 180,E1 -6631.671,E2 -6631.671} C_VEL
LIN {X 0,Y 488.73,Z 373.108,A -85,B 0,C 180,E1 -6634.443,E2 -6634.443} C_VEL
LIN {X 0,Y 488.725,Z 373.104,A -85,B 0,C 180,E1 -6637.153,E2 -6637.153} C_VEL
LIN {X 0,Y 488.732,Z 373.102,A -85,B 0,C 180,E1 -6639.811,E2 -6639.811} C_VEL
LIN {X 0,Y 488.733,Z 373.109,A -85,B 0,C 180,E1 -6642.423,E2 -6642.423} C_VEL
LIN {X 0,Y 488.765,Z 373.099,A -85,B 0,C 180,E1 -6645,E2 -6645} C_VEL
LIN {X 0,Y 488.833,Z 373.098,A -85,B 0,C 180,E1 -6648.388,E2 -6648.388} C_VEL
LIN {X 0,Y 488.789,Z 373.096,A -85,B 0,C 180,E1 -6651.733,E2 -6651.733} C_VEL
LIN {X 0,Y 488.853,Z 373.094,A -85,B 0,C 180,E1 -6654.224,E2 -6654.224} C_VEL
LIN {X 0,Y 488.964,Z 373.073,A -85,B 0,C 180,E1 -6657.529,E2 -6657.529} C_VEL
LIN {X 0,Y 488.958,Z 373.075,A -85,B 0,C 180,E1 -6660.824,E2 -6660.824} C_VEL
LIN {X 0,Y 488.964,Z 373.077,A -85,B 0,C 180,E1 -6662.471,E2 -6662.471} C_VEL
LIN {X 0,Y 488.858,Z 373.09,A -85,B 0,C 180,E1 -6665.776,E2 -6665.776} C_VEL
LIN {X 0,Y 488.819,Z 373.097,A -85,B 0,C 180,E1 -6668.266,E2 -6668.266} C_VEL
LIN {X 0,Y 488.809,Z 373.095,A -85,B 0,C 180,E1 -6671.612,E2 -6671.612} C_VEL
LIN {X 0,Y 488.766,Z 373.097,A -85,B 0,C 180,E1 -6675,E2 -6675} C_VEL
LIN {X 0,Y 488.758,Z 373.1,A -85,B 0,C 180,E1 -6678.442,E2 -6678.442} C_VEL
LIN {X 0,Y 488.711,Z 373.104,A -85,B 0,C 180,E1 -6681.071,E2 -6681.071} C_VEL
LIN {X 0,Y 488.698,Z 373.113,A -85,B 0,C 180,E1 -6683.745,E2 -6683.745} C_VEL
LIN {X 0,Y 488.795,Z 373.094,A -85,B 0,C 180,E1 -6686.944,E2 -6686.944} C_VEL
LIN {X 0,Y 488.713,Z 373.105,A -85,B 0,C 180,E1 -6690.363,E2 -6690.363} C_VEL
LIN {X 0,Y 488.738,Z 373.106,A -85,B 0,C 180,E1 -6693.484,E2 -6693.484} C_VEL
LIN {X 0,Y 488.691,Z 373.107,A -85,B 0,C 180,E1 -6696.356,E2 -6696.356} C_VEL
LIN {X 0,Y 488.704,Z 373.109,A -85,B 0,C 180,E1 -6699.254,E2 -6699.254} C_VEL
LIN {X 0,Y 488.727,Z 373.111,A -85,B 0,C 180,E1 -6701.602,E2 -6701.602} C_VEL
LIN {X 0,Y 488.715,Z 373.104,A -85,B 0,C 180,E1 -6704.801,E2 -6704.801} C_VEL
LIN {X 0,Y 488.694,Z 373.115,A -85,B 0,C 180,E1 -6707.475,E2 -6707.475} C_VEL
LIN {X 0,Y 488.735,Z 373.106,A -85,B 0,C 180,E1 -6709.677,E2 -6709.677} C_VEL
LIN {X 0,Y 488.686,Z 373.109,A -85,B 0,C 180,E1 -6712.842,E2 -6712.842} C_VEL
LIN {X 0,Y 488.738,Z 373.103,A -85,B 0,C 180,E1 -6715.888,E2 -6715.888} C_VEL
LIN {X 0,Y 488.695,Z 373.109,A -85,B 0,C 180,E1 -6718.82,E2 -6718.82} C_VEL
LIN {X 0,Y 488.747,Z 373.103,A -85,B 0,C 180,E1 -6721.671,E2 -6721.671} C_VEL
LIN {X 0,Y 488.745,Z 373.103,A -85,B 0,C 180,E1 -6724.345,E2 -6724.345} C_VEL
LIN {X 0,Y 488.069,Z 373.193,A -85,B 0,C 180,E1 -6725.033,E2 -6725.033} C_VEL
LIN {X 0,Y 485.102,Z 373.561,A -85,B 0,C 180,E1 -6726.148,E2 -6726.148} C_VEL
LIN {X 0,Y 482.657,Z 373.866,A -85,B 0,C 180,E1 -6727.048,E2 -6727.048} C_VEL
LIN {X 0,Y 481.71,Z 373.984,A -85,B 0,C 180,E1 -6727.744,E2 -6727.744} C_VEL
LIN {X 0,Y 481.689,Z 373.986,A -85,B 0,C 180,E1 -6727.979,E2 -6727.979} C_VEL
LIN {X 0,Y 483.038,Z 382.131,A -85,B 0,C 180,E1 -6729.785,E2 -6729.785} C_VEL
LIN {X 0,Y 482.583,Z 394.922,A -85,B 0,C 180,E1 -6732.411,E2 -6732.411} C_VEL
LIN {X 0,Y 482.373,Z 400.542,A -85,B 0,C 180,E1 -6733.543,E2 -6733.543} C_VEL
LIN {X 0,Y 484.993,Z 414.364,A -85,B 0,C 180,E1 -6733.853,E2 -6733.853} C_VEL
LIN {X 0,Y 484.396,Z 507.802,A -85,B 0,C 180,E1 -6735.265,E2 -6735.265} C_VEL
LIN {X 0,Y 484.062,Z 520.933,A -85,B 0,C 180,E1 -6735.63,E2 -6735.63} C_VEL
LIN {X 0,Y 483.707,Z 533.008,A -85,B 0,C 180,E1 -6736.129,E2 -6736.129} C_VEL
LIN {X 0,Y 483.372,Z 544.158,A -85,B 0,C 180,E1 -6736.747,E2 -6736.747} C_VEL
LIN {X 0,Y 482.935,Z 556.07,A -85,B 0,C 180,E1 -6737.605,E2 -6737.605} C_VEL
LIN {X 0,Y 482.455,Z 566.546,A -85,B 0,C 180,E1 -6738.552,E2 -6738.552} C_VEL
LIN {X 0,Y 482.138,Z 575.103,A -85,B 0,C 180,E1 -6739.502,E2 -6739.502} C_VEL
LIN {X 0,Y 481.724,Z 582.987,A -85,B 0,C 180,E1 -6740.553,E2 -6740.553} C_VEL
LIN {X 0,Y 481.407,Z 590.694,A -85,B 0,C 180,E1 -6741.817,E2 -6741.817} C_VEL
LIN {X 0,Y 481.12,Z 597.765,A -85,B 0,C 180,E1 -6743.289,E2 -6743.289} C_VEL
LIN {X 0,Y 481.021,Z 602.475,A -85,B 0,C 180,E1 -6744.551,E2 -6744.551} C_VEL
LIN {X 0,Y 480.938,Z 606.083,A -85,B 0,C 180,E1 -6745.81,E2 -6745.81} C_VEL
LIN {X 0,Y 480.907,Z 607.947,A -85,B 0,C 180,E1 -6746.649,E2 -6746.649} C_VEL
LIN {X 0,Y 480.846,Z 609.354,A -85,B 0,C 180,E1 -6747.487,E2 -6747.487} C_VEL
LIN {X 0,Y 480.823,Z 610.354,A -85,B 0,C 180,E1 -6748.325,E2 -6748.325} C_VEL
LIN {X 0,Y 480.743,Z 611.207,A -85,B 0,C 180,E1 -6750,E2 -6750} C_VEL
LIN {X 0,Y 480.76,Z 611.022,A -85,B 0,C 180,E1 -6750.838,E2 -6750.838} C_VEL
LIN {X 0,Y 480.824,Z 610.437,A -85,B 0,C 180,E1 -6751.675,E2 -6751.675} C_VEL
LIN {X 0,Y 480.907,Z 608.114,A -85,B 0,C 180,E1 -6753.351,E2 -6753.351} C_VEL
LIN {X 0,Y 480.894,Z 605.25,A -85,B 0,C 180,E1 -6754.611,E2 -6754.611} C_VEL
LIN {X 0,Y 481.123,Z 601.361,A -85,B 0,C 180,E1 -6755.869,E2 -6755.869} C_VEL
LIN {X 0,Y 481.196,Z 596.348,A -85,B 0,C 180,E1 -6757.132,E2 -6757.132} C_VEL
LIN {X 0,Y 481.436,Z 590.038,A -85,B 0,C 180,E1 -6758.394,E2 -6758.394} C_VEL
LIN {X 0,Y 481.742,Z 582.136,A -85,B 0,C 180,E1 -6759.658,E2 -6759.658} C_VEL
LIN {X 0,Y 482.098,Z 574.081,A -85,B 0,C 180,E1 -6760.712,E2 -6760.712} C_VEL
LIN {X 0,Y 482.571,Z 564.25,A -85,B 0,C 180,E1 -6761.765,E2 -6761.765} C_VEL
LIN {X 0,Y 482.998,Z 554.579,A -85,B 0,C 180,E1 -6762.607,E2 -6762.607} C_VEL
LIN {X 0,Y 483.345,Z 543.946,A -85,B 0,C 180,E1 -6763.357,E2 -6763.357} C_VEL
LIN {X 0,Y 483.762,Z 531.529,A -85,B 0,C 180,E1 -6764.03,E2 -6764.03} C_VEL
LIN {X 0,Y 484.122,Z 518.933,A -85,B 0,C 180,E1 -6764.529,E2 -6764.529} C_VEL
LIN {X 0,Y 484.355,Z 507.053,A -85,B 0,C 180,E1 -6764.845,E2 -6764.845} C_VEL
LIN {X 0,Y 484.926,Z 413.974,A -85,B 0,C 180,E1 -6766.246,E2 -6766.246} C_VEL
LIN {X 0,Y 482.37,Z 400.518,A -85,B 0,C 180,E1 -6766.549,E2 -6766.549} C_VEL
LIN {X 0,Y 482.974,Z 385.765,A -85,B 0,C 180,E1 -6769.554,E2 -6769.554} C_VEL
LIN {X 0,Y 482.786,Z 379.736,A -85,B 0,C 180,E1 -6770.822,E2 -6770.822} C_VEL
LIN {X 0,Y 481.686,Z 373.987,A -85,B 0,C 180,E1 -6772.124,E2 -6772.124} C_VEL
LIN {X 0,Y 481.715,Z 373.986,A -85,B 0,C 180,E1 -6775.236,E2 -6775.236} C_VEL
LIN {X 0,Y 481.704,Z 373.977,A -85,B 0,C 180,E1 -6777.832,E2 -6777.832} C_VEL
LIN {X 0,Y 481.65,Z 373.991,A -85,B 0,C 180,E1 -6780.711,E2 -6780.711} C_VEL
LIN {X 0,Y 481.701,Z 373.977,A -85,B 0,C 180,E1 -6783.733,E2 -6783.733} C_VEL
LIN {X 0,Y 481.63,Z 373.994,A -85,B 0,C 180,E1 -6786.747,E2 -6786.747} C_VEL
LIN {X 0,Y 481.681,Z 373.981,A -85,B 0,C 180,E1 -6789.941,E2 -6789.941} C_VEL
LIN {X 0,Y 481.643,Z 373.985,A -85,B 0,C 180,E1 -6793.3,E2 -6793.3} C_VEL
LIN {X 0,Y 481.664,Z 373.982,A -85,B 0,C 180,E1 -6795.641,E2 -6795.641} C_VEL
LIN {X 0,Y 481.668,Z 373.984,A -85,B 0,C 180,E1 -6798.959,E2 -6798.959} C_VEL
LIN {X 0,Y 481.659,Z 373.985,A -85,B 0,C 180,E1 -6801.993,E2 -6801.993} C_VEL
LIN {X 0,Y 481.693,Z 373.978,A -85,B 0,C 180,E1 -6805.318,E2 -6805.318} C_VEL
LIN {X 0,Y 481.65,Z 373.992,A -85,B 0,C 180,E1 -6808.312,E2 -6808.312} C_VEL
LIN {X 0,Y 481.705,Z 373.977,A -85,B 0,C 180,E1 -6811.219,E2 -6811.219} C_VEL
LIN {X 0,Y 481.695,Z 373.984,A -85,B 0,C 180,E1 -6814.042,E2 -6814.042} C_VEL
LIN {X 0,Y 481.679,Z 373.981,A -85,B 0,C 180,E1 -6816.812,E2 -6816.812} C_VEL
LIN {X 0,Y 481.703,Z 373.978,A -85,B 0,C 180,E1 -6819.503,E2 -6819.503} C_VEL
LIN {X 0,Y 481.713,Z 373.984,A -85,B 0,C 180,E1 -6822.159,E2 -6822.159} C_VEL
LIN {X 0,Y 481.748,Z 373.972,A -85,B 0,C 180,E1 -6824.776,E2 -6824.776} C_VEL
LIN {X 0,Y 481.757,Z 373.976,A -85,B 0,C 180,E1 -6828.215,E2 -6828.215} C_VEL
LIN {X 0,Y 481.767,Z 373.973,A -85,B 0,C 180,E1 -6831.612,E2 -6831.612} C_VEL
LIN {X 0,Y 481.822,Z 373.968,A -85,B 0,C 180,E1 -6834.14,E2 -6834.14} C_VEL
LIN {X 0,Y 481.934,Z 373.952,A -85,B 0,C 180,E1 -6837.493,E2 -6837.493} C_VEL
LIN {X 0,Y 481.892,Z 373.954,A -85,B 0,C 180,E1 -6840.836,E2 -6840.836} C_VEL
LIN {X 0,Y 481.934,Z 373.949,A -85,B 0,C 180,E1 -6842.507,E2 -6842.507} C_VEL
LIN {X 0,Y 481.821,Z 373.969,A -85,B 0,C 180,E1 -6845.86,E2 -6845.86} C_VEL
LIN {X 0,Y 481.745,Z 373.973,A -85,B 0,C 180,E1 -6848.389,E2 -6848.389} C_VEL
LIN {X 0,Y 481.801,Z 373.971,A -85,B 0,C 180,E1 -6851.784,E2 -6851.784} C_VEL
LIN {X 0,Y 481.748,Z 373.975,A -85,B 0,C 180,E1 -6855.224,E2 -6855.224} C_VEL
LIN {X 0,Y 481.718,Z 373.976,A -85,B 0,C 180,E1 -6858.722,E2 -6858.722} C_VEL
LIN {X 0,Y 481.651,Z 373.991,A -85,B 0,C 180,E1 -6861.394,E2 -6861.394} C_VEL
LIN {X 0,Y 481.666,Z 373.983,A -85,B 0,C 180,E1 -6864.114,E2 -6864.114} C_VEL
LIN {X 0,Y 481.751,Z 373.976,A -85,B 0,C 180,E1 -6867.139,E2 -6867.139} C_VEL
LIN {X 0,Y 481.683,Z 373.983,A -85,B 0,C 180,E1 -6869.741,E2 -6869.741} C_VEL
LIN {X 0,Y 481.674,Z 373.982,A -85,B 0,C 180,E1 -6872.674,E2 -6872.674} C_VEL
LIN {X 0,Y 481.64,Z 373.988,A -85,B 0,C 180,E1 -6875.709,E2 -6875.709} C_VEL
LIN {X 0,Y 481.674,Z 373.984,A -85,B 0,C 180,E1 -6878.859,E2 -6878.859} C_VEL
LIN {X 0,Y 481.656,Z 373.983,A -85,B 0,C 180,E1 -6881.913,E2 -6881.913} C_VEL
LIN {X 0,Y 481.664,Z 373.983,A -85,B 0,C 180,E1 -6884.457,E2 -6884.457} C_VEL
LIN {X 0,Y 481.651,Z 373.984,A -85,B 0,C 180,E1 -6887.839,E2 -6887.839} C_VEL
LIN {X 0,Y 481.685,Z 373.983,A -85,B 0,C 180,E1 -6890.651,E2 -6890.651} C_VEL
LIN {X 0,Y 481.631,Z 373.989,A -85,B 0,C 180,E1 -6893.376,E2 -6893.376} C_VEL
LIN {X 0,Y 481.713,Z 373.977,A -85,B 0,C 180,E1 -6896.33,E2 -6896.33} C_VEL
LIN {X 0,Y 481.654,Z 373.988,A -85,B 0,C 180,E1 -6899.417,E2 -6899.417} C_VEL
LIN {X 0,Y 481.704,Z 373.982,A -85,B 0,C 180,E1 -6902.168,E2 -6902.168} C_VEL
LIN {X 0,Y 481.74,Z 374.151,A -85,B 0,C 180,E1 -6904.971,E2 -6904.971} C_VEL
LIN {X 0,Y 483.641,Z 384.176,A -85,B 0,C 180,E1 -6906.899,E2 -6906.899} C_VEL
LIN {X 0,Y 483.327,Z 395.414,A -85,B 0,C 180,E1 -6908.906,E2 -6908.906} C_VEL
LIN {X 0,Y 482.577,Z 414.1,A -85,B 0,C 180,E1 -6912.191,E2 -6912.191} C_VEL
LIN {X 0,Y 482.329,Z 421.496,A -85,B 0,C 180,E1 -6913.486,E2 -6913.486} C_VEL
LIN {X 0,Y 484.916,Z 438.43,A -85,B 0,C 180,E1 -6913.837,E2 -6913.837} C_VEL
LIN {X 0,Y 484.289,Z 529.489,A -85,B 0,C 180,E1 -6915.207,E2 -6915.207} C_VEL
LIN {X 0,Y 483.978,Z 542.772,A -85,B 0,C 180,E1 -6915.574,E2 -6915.574} C_VEL
LIN {X 0,Y 483.54,Z 554.938,A -85,B 0,C 180,E1 -6916.07,E2 -6916.07} C_VEL
LIN {X 0,Y 483.147,Z 567.218,A -85,B 0,C 180,E1 -6916.756,E2 -6916.756} C_VEL
LIN {X 0,Y 482.73,Z 577.135,A -85,B 0,C 180,E1 -6917.461,E2 -6917.461} C_VEL
LIN {X 0,Y 482.301,Z 588.183,A -85,B 0,C 180,E1 -6918.442,E2 -6918.442} C_VEL
LIN {X 0,Y 481.872,Z 597.792,A -85,B 0,C 180,E1 -6919.495,E2 -6919.495} C_VEL
LIN {X 0,Y 481.531,Z 605.668,A -85,B 0,C 180,E1 -6920.549,E2 -6920.549} C_VEL
LIN {X 0,Y 481.251,Z 613.361,A -85,B 0,C 180,E1 -6921.814,E2 -6921.814} C_VEL
LIN {X 0,Y 481.02,Z 620.452,A -85,B 0,C 180,E1 -6923.287,E2 -6923.287} C_VEL
LIN {X 0,Y 480.949,Z 625.171,A -85,B 0,C 180,E1 -6924.549,E2 -6924.549} C_VEL
LIN {X 0,Y 480.828,Z 628.774,A -85,B 0,C 180,E1 -6925.809,E2 -6925.809} C_VEL
LIN {X 0,Y 480.87,Z 630.635,A -85,B 0,C 180,E1 -6926.648,E2 -6926.648} C_VEL
LIN {X 0,Y 480.823,Z 632.029,A -85,B 0,C 180,E1 -6927.487,E2 -6927.487} C_VEL
LIN {X 0,Y 480.76,Z 633.63,A -85,B 0,C 180,E1 -6929.162,E2 -6929.162} C_VEL
LIN {X 0,Y 480.743,Z 633.846,A -85,B 0,C 180,E1 -6930,E2 -6930} C_VEL
LIN {X 0,Y 480.792,Z 633.025,A -85,B 0,C 180,E1 -6931.675,E2 -6931.675} C_VEL
LIN {X 0,Y 480.823,Z 632.032,A -85,B 0,C 180,E1 -6932.513,E2 -6932.513} C_VEL
LIN {X 0,Y 480.87,Z 630.639,A -85,B 0,C 180,E1 -6933.351,E2 -6933.351} C_VEL
LIN {X 0,Y 480.84,Z 627.706,A -85,B 0,C 180,E1 -6934.611,E2 -6934.611} C_VEL
LIN {X 0,Y 480.965,Z 623.739,A -85,B 0,C 180,E1 -6935.871,E2 -6935.871} C_VEL
LIN {X 0,Y 481.112,Z 617.636,A -85,B 0,C 180,E1 -6937.343,E2 -6937.343} C_VEL
LIN {X 0,Y 481.328,Z 610.966,A -85,B 0,C 180,E1 -6938.607,E2 -6938.607} C_VEL
LIN {X 0,Y 481.664,Z 602.69,A -85,B 0,C 180,E1 -6939.872,E2 -6939.872} C_VEL
LIN {X 0,Y 482.041,Z 594.208,A -85,B 0,C 180,E1 -6940.926,E2 -6940.926} C_VEL
LIN {X 0,Y 482.521,Z 583.727,A -85,B 0,C 180,E1 -6941.979,E2 -6941.979} C_VEL
LIN {X 0,Y 482.878,Z 572.426,A -85,B 0,C 180,E1 -6942.893,E2 -6942.893} C_VEL
LIN {X 0,Y 483.361,Z 560.065,A -85,B 0,C 180,E1 -6943.667,E2 -6943.667} C_VEL
LIN {X 0,Y 483.776,Z 547.723,A -85,B 0,C 180,E1 -6944.244,E2 -6944.244} C_VEL
LIN {X 0,Y 484.142,Z 535.059,A -85,B 0,C 180,E1 -6944.663,E2 -6944.663} C_VEL
LIN {X 0,Y 484.384,Z 521.841,A -85,B 0,C 180,E1 -6944.924,E2 -6944.924} C_VEL
LIN {X 0,Y 484.821,Z 437.141,A -85,B 0,C 180,E1 -6946.185,E2 -6946.185} C_VEL
LIN {X 0,Y 482.35,Z 421.52,A -85,B 0,C 180,E1 -6946.507,E2 -6946.507} C_VEL
LIN {X 0,Y 482.934,Z 404.137,A -85,B 0,C 180,E1 -6949.555,E2 -6949.555} C_VEL
LIN {X 0,Y 483.705,Z 386.67,A -85,B 0,C 180,E1 -6952.646,E2 -6952.646} C_VEL
LIN {X 0,Y 483.327,Z 382.241,A -85,B 0,C 180,E1 -6953.465,E2 -6953.465} C_VEL
LIN {X 0,Y 481.72,Z 373.982,A -85,B 0,C 180,E1 -6955.088,E2 -6955.088} C_VEL
LIN {X 0,Y 481.703,Z 373.982,A -85,B 0,C 180,E1 -6957.832,E2 -6957.832} C_VEL
LIN {X 0,Y 481.649,Z 373.987,A -85,B 0,C 180,E1 -6960.711,E2 -6960.711} C_VEL
LIN {X 0,Y 481.699,Z 373.979,A -85,B 0,C 180,E1 -6963.733,E2 -6963.733} C_VEL
LIN {X 0,Y 481.628,Z 373.991,A -85,B 0,C 180,E1 -6966.747,E2 -6966.747} C_VEL
LIN {X 0,Y 481.679,Z 373.98,A -85,B 0,C 180,E1 -6969.94,E2 -6969.94} C_VEL
LIN {X 0,Y 481.641,Z 373.988,A -85,B 0,C 180,E1 -6973.3,E2 -6973.3} C_VEL
LIN {X 0,Y 481.661,Z 373.983,A -85,B 0,C 180,E1 -6975.641,E2 -6975.641} C_VEL
LIN {X 0,Y 481.665,Z 373.989,A -85,B 0,C 180,E1 -6978.959,E2 -6978.959} C_VEL
LIN {X 0,Y 481.657,Z 373.983,A -85,B 0,C 180,E1 -6981.993,E2 -6981.993} C_VEL
LIN {X 0,Y 481.69,Z 373.98,A -85,B 0,C 180,E1 -6985.318,E2 -6985.318} C_VEL
LIN {X 0,Y 481.647,Z 373.987,A -85,B 0,C 180,E1 -6988.312,E2 -6988.312} C_VEL
LIN {X 0,Y 481.703,Z 373.979,A -85,B 0,C 180,E1 -6991.219,E2 -6991.219} C_VEL
LIN {X 0,Y 481.692,Z 373.98,A -85,B 0,C 180,E1 -6994.042,E2 -6994.042} C_VEL
LIN {X 0,Y 481.676,Z 373.986,A -85,B 0,C 180,E1 -6996.812,E2 -6996.812} C_VEL
LIN {X 0,Y 481.7,Z 373.977,A -85,B 0,C 180,E1 -6999.503,E2 -6999.503} C_VEL
LIN {X 0,Y 481.707,Z 373.98,A -85,B 0,C 180,E1 -7002.158,E2 -7002.158} C_VEL
LIN {X 0,Y 481.746,Z 373.976,A -85,B 0,C 180,E1 -7004.776,E2 -7004.776} C_VEL
LIN {X 0,Y 481.798,Z 373.971,A -85,B 0,C 180,E1 -7008.216,E2 -7008.216} C_VEL
LIN {X 0,Y 481.744,Z 373.973,A -85,B 0,C 180,E1 -7011.611,E2 -7011.611} C_VEL
LIN {X 0,Y 481.814,Z 373.97,A -85,B 0,C 180,E1 -7014.14,E2 -7014.14} C_VEL
LIN {X 0,Y 481.931,Z 373.949,A -85,B 0,C 180,E1 -7017.493,E2 -7017.493} C_VEL
LIN {X 0,Y 481.909,Z 373.953,A -85,B 0,C 180,E1 -7020.836,E2 -7020.836} C_VEL
LIN {X 0,Y 481.931,Z 373.953,A -85,B 0,C 180,E1 -7022.507,E2 -7022.507} C_VEL
LIN {X 0,Y 481.819,Z 373.967,A -85,B 0,C 180,E1 -7025.86,E2 -7025.86} C_VEL
LIN {X 0,Y 481.765,Z 373.974,A -85,B 0,C 180,E1 -7028.388,E2 -7028.388} C_VEL
LIN {X 0,Y 481.754,Z 373.976,A -85,B 0,C 180,E1 -7031.785,E2 -7031.785} C_VEL
LIN {X 0,Y 481.746,Z 373.972,A -85,B 0,C 180,E1 -7035.224,E2 -7035.224} C_VEL
LIN {X 0,Y 481.716,Z 373.976,A -85,B 0,C 180,E1 -7038.722,E2 -7038.722} C_VEL
LIN {X 0,Y 481.65,Z 373.986,A -85,B 0,C 180,E1 -7041.395,E2 -7041.395} C_VEL
LIN {X 0,Y 481.681,Z 373.984,A -85,B 0,C 180,E1 -7044.113,E2 -7044.113} C_VEL
LIN {X 0,Y 481.75,Z 373.972,A -85,B 0,C 180,E1 -7047.139,E2 -7047.139} C_VEL
LIN {X 0,Y 481.682,Z 373.988,A -85,B 0,C 180,E1 -7049.741,E2 -7049.741} C_VEL
LIN {X 0,Y 481.675,Z 373.981,A -85,B 0,C 180,E1 -7052.674,E2 -7052.674} C_VEL
LIN {X 0,Y 481.645,Z 373.992,A -85,B 0,C 180,E1 -7055.709,E2 -7055.709} C_VEL
LIN {X 0,Y 481.673,Z 373.981,A -85,B 0,C 180,E1 -7058.859,E2 -7058.859} C_VEL
LIN {X 0,Y 481.665,Z 373.986,A -85,B 0,C 180,E1 -7061.914,E2 -7061.914} C_VEL
LIN {X 0,Y 481.663,Z 373.982,A -85,B 0,C 180,E1 -7064.457,E2 -7064.457} C_VEL
LIN {X 0,Y 481.65,Z 373.987,A -85,B 0,C 180,E1 -7067.839,E2 -7067.839} C_VEL
LIN {X 0,Y 481.683,Z 373.98,A -85,B 0,C 180,E1 -7070.651,E2 -7070.651} C_VEL
LIN {X 0,Y 481.635,Z 373.994,A -85,B 0,C 180,E1 -7073.375,E2 -7073.375} C_VEL
LIN {X 0,Y 481.712,Z 373.976,A -85,B 0,C 180,E1 -7076.33,E2 -7076.33} C_VEL
LIN {X 0,Y 481.654,Z 373.99,A -85,B 0,C 180,E1 -7079.417,E2 -7079.417} C_VEL
LIN {X 0,Y 481.703,Z 373.977,A -85,B 0,C 180,E1 -7082.168,E2 -7082.168} C_VEL
LIN {X 0,Y 481.72,Z 373.983,A -85,B 0,C 180,E1 -7084.97,E2 -7084.97} C_VEL
LIN {X 0,Y 481.689,Z 373.986,A -85,B 0,C 180,E1 -7087.979,E2 -7087.979} C_VEL
LIN {X 0,Y 481.316,Z 377.165,A -85,B 0,C 180,E1 -7088.656,E2 -7088.656} C_VEL
LIN {X 0,Y 479.04,Z 382.294,A -85,B 0,C 180,E1 -7089.625,E2 -7089.625} C_VEL
LIN {X 0,Y 476.557,Z 387.475,A -85,B 0,C 180,E1 -7090.561,E2 -7090.561} C_VEL
LIN {X 0,Y 475.834,Z 390.327,A -85,B 0,C 180,E1 -7091.163,E2 -7091.163} C_VEL
LIN {X 0,Y 475.415,Z 400.733,A -85,B 0,C 180,E1 -7093.3,E2 -7093.3} C_VEL
LIN {X 0,Y 478.199,Z 415.944,A -85,B 0,C 180,E1 -7093.639,E2 -7093.639} C_VEL
LIN {X 0,Y 477.555,Z 507.989,A -85,B 0,C 180,E1 -7095.049,E2 -7095.049} C_VEL
LIN {X 0,Y 477.187,Z 521.114,A -85,B 0,C 180,E1 -7095.419,E2 -7095.419} C_VEL
LIN {X 0,Y 476.824,Z 533.185,A -85,B 0,C 180,E1 -7095.925,E2 -7095.925} C_VEL
LIN {X 0,Y 476.46,Z 544.546,A -85,B 0,C 180,E1 -7096.565,E2 -7096.565} C_VEL
LIN {X 0,Y 476.01,Z 556.243,A -85,B 0,C 180,E1 -7097.422,E2 -7097.422} C_VEL
LIN {X 0,Y 475.502,Z 566.718,A -85,B 0,C 180,E1 -7098.382,E2 -7098.382} C_VEL
LIN {X 0,Y 475.148,Z 575.274,A -85,B 0,C 180,E1 -7099.345,E2 -7099.345} C_VEL
LIN {X 0,Y 474.721,Z 583.158,A -85,B 0,C 180,E1 -7100.413,E2 -7100.413} C_VEL
LIN {X 0,Y 474.371,Z 590.864,A -85,B 0,C 180,E1 -7101.695,E2 -7101.695} C_VEL
LIN {X 0,Y 474.069,Z 597.934,A -85,B 0,C 180,E1 -7103.189,E2 -7103.189} C_VEL
LIN {X 0,Y 473.971,Z 602.643,A -85,B 0,C 180,E1 -7104.469,E2 -7104.469} C_VEL
LIN {X 0,Y 473.84,Z 606.251,A -85,B 0,C 180,E1 -7105.747,E2 -7105.747} C_VEL
LIN {X 0,Y 473.837,Z 608.115,A -85,B 0,C 180,E1 -7106.599,E2 -7106.599} C_VEL
LIN {X 0,Y 473.763,Z 609.522,A -85,B 0,C 180,E1 -7107.449,E2 -7107.449} C_VEL
LIN {X 0,Y 473.689,Z 611.138,A -85,B 0,C 180,E1 -7109.15,E2 -7109.15} C_VEL
LIN {X 0,Y 473.67,Z 611.374,A -85,B 0,C 180,E1 -7110,E2 -7110} C_VEL
LIN {X 0,Y 473.689,Z 611.188,A -85,B 0,C 180,E1 -7110.85,E2 -7110.85} C_VEL
LIN {X 0,Y 473.763,Z 609.637,A -85,B 0,C 180,E1 -7112.551,E2 -7112.551} C_VEL
LIN {X 0,Y 473.837,Z 608.28,A -85,B 0,C 180,E1 -7113.401,E2 -7113.401} C_VEL
LIN {X 0,Y 473.809,Z 605.416,A -85,B 0,C 180,E1 -7114.68,E2 -7114.68} C_VEL
LIN {X 0,Y 474.043,Z 601.526,A -85,B 0,C 180,E1 -7115.957,E2 -7115.957} C_VEL
LIN {X 0,Y 474.146,Z 596.513,A -85,B 0,C 180,E1 -7117.238,E2 -7117.238} C_VEL
LIN {X 0,Y 474.407,Z 590.202,A -85,B 0,C 180,E1 -7118.52,E2 -7118.52} C_VEL
LIN {X 0,Y 474.729,Z 582.3,A -85,B 0,C 180,E1 -7119.803,E2 -7119.803} C_VEL
LIN {X 0,Y 475.099,Z 574.245,A -85,B 0,C 180,E1 -7120.872,E2 -7120.872} C_VEL
LIN {X 0,Y 475.624,Z 564.412,A -85,B 0,C 180,E1 -7121.939,E2 -7121.939} C_VEL
LIN {X 0,Y 476.097,Z 553.604,A -85,B 0,C 180,E1 -7122.883,E2 -7122.883} C_VEL
LIN {X 0,Y 476.509,Z 542.524,A -85,B 0,C 180,E1 -7123.65,E2 -7123.65} C_VEL
LIN {X 0,Y 476.931,Z 530.558,A -85,B 0,C 180,E1 -7124.29,E2 -7124.29} C_VEL
LIN {X 0,Y 477.301,Z 518.311,A -85,B 0,C 180,E1 -7124.769,E2 -7124.769} C_VEL
LIN {X 0,Y 477.548,Z 505.757,A -85,B 0,C 180,E1 -7125.088,E2 -7125.088} C_VEL
LIN {X 0,Y 478.025,Z 414.399,A -85,B 0,C 180,E1 -7126.483,E2 -7126.483} C_VEL
LIN {X 0,Y 475.395,Z 400.678,A -85,B 0,C 180,E1 -7126.799,E2 -7126.799} C_VEL
LIN {X 0,Y 475.992,Z 385.908,A -85,B 0,C 180,E1 -7129.852,E2 -7129.852} C_VEL
LIN {X 0,Y 475.905,Z 381.652,A -85,B 0,C 180,E1 -7130.758,E2 -7130.758} C_VEL
LIN {X 0,Y 474.639,Z 374.866,A -85,B 0,C 180,E1 -7132.299,E2 -7132.299} C_VEL
LIN {X 0,Y 474.675,Z 374.861,A -85,B 0,C 180,E1 -7135.428,E2 -7135.428} C_VEL
LIN {X 0,Y 474.65,Z 374.858,A -85,B 0,C 180,E1 -7138.283,E2 -7138.283} C_VEL
LIN {X 0,Y 474.603,Z 374.864,A -85,B 0,C 180,E1 -7141.218,E2 -7141.218} C_VEL
LIN {X 0,Y 474.636,Z 374.86,A -85,B 0,C 180,E1 -7144.241,E2 -7144.241} C_VEL
LIN {X 0,Y 474.594,Z 374.864,A -85,B 0,C 180,E1 -7147.384,E2 -7147.384} C_VEL
LIN {X 0,Y 474.621,Z 374.868,A -85,B 0,C 180,E1 -7150.658,E2 -7150.658} C_VEL
LIN {X 0,Y 474.606,Z 374.861,A -85,B 0,C 180,E1 -7153.481,E2 -7153.481} C_VEL
LIN {X 0,Y 474.627,Z 374.867,A -85,B 0,C 180,E1 -7156.516,E2 -7156.516} C_VEL
LIN {X 0,Y 474.624,Z 374.859,A -85,B 0,C 180,E1 -7159.343,E2 -7159.343} C_VEL
LIN {X 0,Y 474.614,Z 374.861,A -85,B 0,C 180,E1 -7161.704,E2 -7161.704} C_VEL
LIN {X 0,Y 474.629,Z 374.862,A -85,B 0,C 180,E1 -7164.726,E2 -7164.726} C_VEL
LIN {X 0,Y 474.64,Z 374.859,A -85,B 0,C 180,E1 -7167.788,E2 -7167.788} C_VEL
LIN {X 0,Y 474.629,Z 374.86,A -85,B 0,C 180,E1 -7170.885,E2 -7170.885} C_VEL
LIN {X 0,Y 474.659,Z 374.856,A -85,B 0,C 180,E1 -7173.628,E2 -7173.628} C_VEL
LIN {X 0,Y 474.64,Z 374.86,A -85,B 0,C 180,E1 -7176.642,E2 -7176.642} C_VEL
LIN {X 0,Y 474.663,Z 374.862,A -85,B 0,C 180,E1 -7180.09,E2 -7180.09} C_VEL
LIN {X 0,Y 474.656,Z 374.856,A -85,B 0,C 180,E1 -7182.775,E2 -7182.775} C_VEL
LIN {X 0,Y 474.654,Z 374.856,A -85,B 0,C 180,E1 -7185.421,E2 -7185.421} C_VEL
LIN {X 0,Y 474.711,Z 374.857,A -85,B 0,C 180,E1 -7188.038,E2 -7188.038} C_VEL
LIN {X 0,Y 474.732,Z 374.848,A -85,B 0,C 180,E1 -7191.486,E2 -7191.486} C_VEL
LIN {X 0,Y 474.785,Z 374.846,A -85,B 0,C 180,E1 -7194.052,E2 -7194.052} C_VEL
LIN {X 0,Y 474.9,Z 374.828,A -85,B 0,C 180,E1 -7197.455,E2 -7197.455} C_VEL
LIN {X 0,Y 474.918,Z 374.828,A -85,B 0,C 180,E1 -7200,E2 -7200} C_VEL
LIN {X 0,Y 474.9,Z 374.825,A -85,B 0,C 180,E1 -7202.545,E2 -7202.545} C_VEL
LIN {X 0,Y 474.784,Z 374.844,A -85,B 0,C 180,E1 -7205.948,E2 -7205.948} C_VEL
LIN {X 0,Y 474.716,Z 374.848,A -85,B 0,C 180,E1 -7208.514,E2 -7208.514} C_VEL
LIN {X 0,Y 474.745,Z 374.848,A -85,B 0,C 180,E1 -7211.961,E2 -7211.961} C_VEL
LIN {X 0,Y 474.686,Z 374.857,A -85,B 0,C 180,E1 -7215.768,E2 -7215.768} C_VEL
LIN {X 0,Y 474.671,Z 374.855,A -85,B 0,C 180,E1 -7219.01,E2 -7219.01} C_VEL
LIN {X 0,Y 474.594,Z 374.868,A -85,B 0,C 180,E1 -7221.729,E2 -7221.729} C_VEL
LIN {X 0,Y 474.646,Z 374.856,A -85,B 0,C 180,E1 -7224.494,E2 -7224.494} C_VEL
LIN {X 0,Y 474.686,Z 374.859,A -85,B 0,C 180,E1 -7227.334,E2 -7227.334} C_VEL
LIN {X 0,Y 474.61,Z 374.861,A -85,B 0,C 180,E1 -7230.23,E2 -7230.23} C_VEL
LIN {X 0,Y 474.629,Z 374.866,A -85,B 0,C 180,E1 -7233.221,E2 -7233.221} C_VEL
LIN {X 0,Y 474.592,Z 374.863,A -85,B 0,C 180,E1 -7236.323,E2 -7236.323} C_VEL
LIN {X 0,Y 474.622,Z 374.862,A -85,B 0,C 180,E1 -7239.646,E2 -7239.646} C_VEL
LIN {X 0,Y 474.636,Z 374.863,A -85,B 0,C 180,E1 -7242.932,E2 -7242.932} C_VEL
LIN {X 0,Y 474.613,Z 374.861,A -85,B 0,C 180,E1 -7245.895,E2 -7245.895} C_VEL
LIN {X 0,Y 474.631,Z 374.867,A -85,B 0,C 180,E1 -7249.041,E2 -7249.041} C_VEL
LIN {X 0,Y 474.614,Z 374.861,A -85,B 0,C 180,E1 -7251.704,E2 -7251.704} C_VEL
LIN {X 0,Y 474.629,Z 374.864,A -85,B 0,C 180,E1 -7254.726,E2 -7254.726} C_VEL
LIN {X 0,Y 474.639,Z 374.857,A -85,B 0,C 180,E1 -7257.788,E2 -7257.788} C_VEL
LIN {X 0,Y 474.628,Z 374.867,A -85,B 0,C 180,E1 -7260.884,E2 -7260.884} C_VEL
LIN {X 0,Y 474.664,Z 374.86,A -85,B 0,C 180,E1 -7263.628,E2 -7263.628} C_VEL
LIN {X 0,Y 474.674,Z 374.9,A -85,B 0,C 180,E1 -7264.739,E2 -7264.739} C_VEL
LIN {X 0,Y 476.777,Z 386.535,A -85,B 0,C 180,E1 -7267.006,E2 -7267.006} C_VEL
LIN {X 0,Y 476.034,Z 403.999,A -85,B 0,C 180,E1 -7270.149,E2 -7270.149} C_VEL
LIN {X 0,Y 475.381,Z 421.54,A -85,B 0,C 180,E1 -7273.246,E2 -7273.246} C_VEL
LIN {X 0,Y 478.101,Z 439.262,A -85,B 0,C 180,E1 -7273.615,E2 -7273.615} C_VEL
LIN {X 0,Y 477.437,Z 529.33,A -85,B 0,C 180,E1 -7274.99,E2 -7274.99} C_VEL
LIN {X 0,Y 477.117,Z 542.61,A -85,B 0,C 180,E1 -7275.362,E2 -7275.362} C_VEL
LIN {X 0,Y 476.645,Z 554.775,A -85,B 0,C 180,E1 -7275.865,E2 -7275.865} C_VEL
LIN {X 0,Y 476.226,Z 567.054,A -85,B 0,C 180,E1 -7276.56,E2 -7276.56} C_VEL
LIN {X 0,Y 475.743,Z 577.837,A -85,B 0,C 180,E1 -7277.346,E2 -7277.346} C_VEL
LIN {X 0,Y 475.281,Z 589.089,A -85,B 0,C 180,E1 -7278.377,E2 -7278.377} C_VEL
LIN {X 0,Y 474.863,Z 597.625,A -85,B 0,C 180,E1 -7279.339,E2 -7279.339} C_VEL
LIN {X 0,Y 474.489,Z 605.501,A -85,B 0,C 180,E1 -7280.408,E2 -7280.408} C_VEL
LIN {X 0,Y 474.177,Z 613.193,A -85,B 0,C 180,E1 -7281.691,E2 -7281.691} C_VEL
LIN {X 0,Y 473.937,Z 620.285,A -85,B 0,C 180,E1 -7283.187,E2 -7283.187} C_VEL
LIN {X 0,Y 473.866,Z 625.004,A -85,B 0,C 180,E1 -7284.468,E2 -7284.468} C_VEL
LIN {X 0,Y 473.735,Z 628.607,A -85,B 0,C 180,E1 -7285.746,E2 -7285.746} C_VEL
LIN {X 0,Y 473.765,Z 630.468,A -85,B 0,C 180,E1 -7286.598,E2 -7286.598} C_VEL
LIN {X 0,Y 473.74,Z 631.862,A -85,B 0,C 180,E1 -7287.449,E2 -7287.449} C_VEL
LIN {X 0,Y 473.688,Z 633.463,A -85,B 0,C 180,E1 -7289.15,E2 -7289.15} C_VEL
LIN {X 0,Y 473.669,Z 633.679,A -85,B 0,C 180,E1 -7290,E2 -7290} C_VEL
LIN {X 0,Y 473.688,Z 633.464,A -85,B 0,C 180,E1 -7290.85,E2 -7290.85} C_VEL
LIN {X 0,Y 473.74,Z 631.865,A -85,B 0,C 180,E1 -7292.551,E2 -7292.551} C_VEL
LIN {X 0,Y 473.765,Z 630.472,A -85,B 0,C 180,E1 -7293.402,E2 -7293.402} C_VEL
LIN {X 0,Y 473.764,Z 627.539,A -85,B 0,C 180,E1 -7294.68,E2 -7294.68} C_VEL
LIN {X 0,Y 473.866,Z 623.571,A -85,B 0,C 180,E1 -7295.959,E2 -7295.959} C_VEL
LIN {X 0,Y 474.031,Z 617.468,A -85,B 0,C 180,E1 -7297.454,E2 -7297.454} C_VEL
LIN {X 0,Y 474.291,Z 610.798,A -85,B 0,C 180,E1 -7298.736,E2 -7298.736} C_VEL
LIN {X 0,Y 474.617,Z 602.521,A -85,B 0,C 180,E1 -7300.02,E2 -7300.02} C_VEL
LIN {X 0,Y 475.05,Z 594.039,A -85,B 0,C 180,E1 -7301.088,E2 -7301.088} C_VEL
LIN {X 0,Y 475.552,Z 583.75,A -85,B 0,C 180,E1 -7302.139,E2 -7302.139} C_VEL
LIN {X 0,Y 475.894,Z 573.473,A -85,B 0,C 180,E1 -7302.993,E2 -7302.993} C_VEL
LIN {X 0,Y 476.383,Z 561.816,A -85,B 0,C 180,E1 -7303.762,E2 -7303.762} C_VEL
LIN {X 0,Y 476.81,Z 550.155,A -85,B 0,C 180,E1 -7304.348,E2 -7304.348} C_VEL
LIN {X 0,Y 477.226,Z 536.716,A -85,B 0,C 180,E1 -7304.826,E2 -7304.826} C_VEL
LIN {X 0,Y 477.524,Z 523.438,A -85,B 0,C 180,E1 -7305.116,E2 -7305.116} C_VEL
LIN {X 0,Y 477.94,Z 437.739,A -85,B 0,C 180,E1 -7306.413,E2 -7306.413} C_VEL
LIN {X 0,Y 475.35,Z 421.354,A -85,B 0,C 180,E1 -7306.757,E2 -7306.757} C_VEL
LIN {X 0,Y 476.031,Z 403.984,A -85,B 0,C 180,E1 -7309.85,E2 -7309.85} C_VEL
LIN {X 0,Y 476.781,Z 386.525,A -85,B 0,C 180,E1 -7312.993,E2 -7312.993} C_VEL
LIN {X 0,Y 474.689,Z 374.857,A -85,B 0,C 180,E1 -7315.278,E2 -7315.278} C_VEL
LIN {X 0,Y 474.649,Z 374.86,A -85,B 0,C 180,E1 -7318.282,E2 -7318.282} C_VEL
LIN {X 0,Y 474.603,Z 374.869,A -85,B 0,C 180,E1 -7321.217,E2 -7321.217} C_VEL
LIN {X 0,Y 474.634,Z 374.858,A -85,B 0,C 180,E1 -7324.241,E2 -7324.241} C_VEL
LIN {X 0,Y 474.592,Z 374.867,A -85,B 0,C 180,E1 -7327.384,E2 -7327.384} C_VEL
LIN {X 0,Y 474.63,Z 374.859,A -85,B 0,C 180,E1 -7329.648,E2 -7329.648} C_VEL
LIN {X 0,Y 474.617,Z 374.868,A -85,B 0,C 180,E1 -7332.934,E2 -7332.934} C_VEL
LIN {X 0,Y 474.617,Z 374.86,A -85,B 0,C 180,E1 -7335.896,E2 -7335.896} C_VEL
LIN {X 0,Y 474.634,Z 374.863,A -85,B 0,C 180,E1 -7339.04,E2 -7339.04} C_VEL
LIN {X 0,Y 474.612,Z 374.861,A -85,B 0,C 180,E1 -7341.704,E2 -7341.704} C_VEL
LIN {X 0,Y 474.627,Z 374.867,A -85,B 0,C 180,E1 -7344.726,E2 -7344.726} C_VEL
LIN {X 0,Y 474.638,Z 374.857,A -85,B 0,C 180,E1 -7347.788,E2 -7347.788} C_VEL
LIN {X 0,Y 474.627,Z 374.864,A -85,B 0,C 180,E1 -7350.884,E2 -7350.884} C_VEL
LIN {X 0,Y 474.656,Z 374.855,A -85,B 0,C 180,E1 -7353.628,E2 -7353.628} C_VEL
LIN {X 0,Y 474.637,Z 374.865,A -85,B 0,C 180,E1 -7356.642,E2 -7356.642} C_VEL
LIN {X 0,Y 474.659,Z 374.857,A -85,B 0,C 180,E1 -7360.09,E2 -7360.09} C_VEL
LIN {X 0,Y 474.651,Z 374.86,A -85,B 0,C 180,E1 -7362.774,E2 -7362.774} C_VEL
LIN {X 0,Y 474.651,Z 374.856,A -85,B 0,C 180,E1 -7365.421,E2 -7365.421} C_VEL
LIN {X 0,Y 474.742,Z 374.848,A -85,B 0,C 180,E1 -7368.039,E2 -7368.039} C_VEL
LIN {X 0,Y 474.715,Z 374.848,A -85,B 0,C 180,E1 -7371.486,E2 -7371.486} C_VEL
LIN {X 0,Y 474.776,Z 374.845,A -85,B 0,C 180,E1 -7374.052,E2 -7374.052} C_VEL
LIN {X 0,Y 474.897,Z 374.825,A -85,B 0,C 180,E1 -7377.455,E2 -7377.455} C_VEL
LIN {X 0,Y 474.915,Z 374.828,A -85,B 0,C 180,E1 -7380,E2 -7380} C_VEL
LIN {X 0,Y 474.897,Z 374.828,A -85,B 0,C 180,E1 -7382.545,E2 -7382.545} C_VEL
LIN {X 0,Y 474.782,Z 374.845,A -85,B 0,C 180,E1 -7385.948,E2 -7385.948} C_VEL
LIN {X 0,Y 474.73,Z 374.849,A -85,B 0,C 180,E1 -7388.514,E2 -7388.514} C_VEL
LIN {X 0,Y 474.708,Z 374.856,A -85,B 0,C 180,E1 -7391.962,E2 -7391.962} C_VEL
LIN {X 0,Y 474.703,Z 374.851,A -85,B 0,C 180,E1 -7395.456,E2 -7395.456} C_VEL
LIN {X 0,Y 474.669,Z 374.853,A -85,B 0,C 180,E1 -7399.01,E2 -7399.01} C_VEL
LIN {X 0,Y 474.595,Z 374.869,A -85,B 0,C 180,E1 -7401.729,E2 -7401.729} C_VEL
LIN {X 0,Y 474.663,Z 374.855,A -85,B 0,C 180,E1 -7404.493,E2 -7404.493} C_VEL
LIN {X 0,Y 474.702,Z 374.852,A -85,B 0,C 180,E1 -7407.339,E2 -7407.339} C_VEL
LIN {X 0,Y 474.607,Z 374.861,A -85,B 0,C 180,E1 -7410.81,E2 -7410.81} C_VEL
